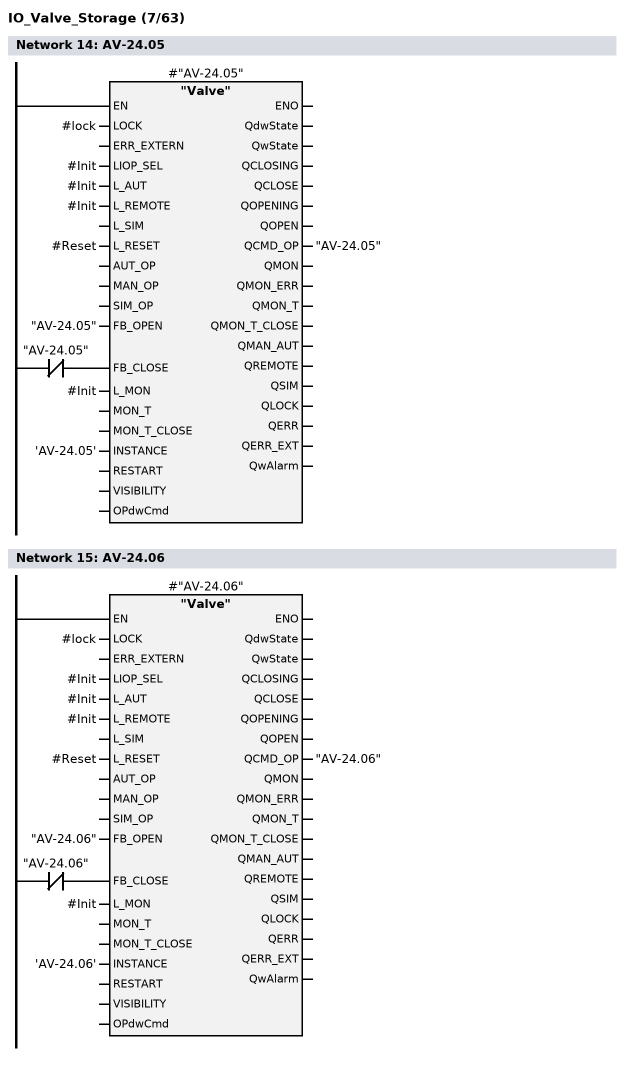
   RUNG wire#powerrail
      #"AV-24.05"(FB_CLOSE := wire#w1, LOCK := #lock, ERR_EXTERN :=, LIOP_SEL := #Init, L_AUT := #Init, L_REMOTE := #Init, L_SIM :=, L_RESET := #Reset, AUT_OP :=, MAN_OP :=, SIM_OP :=, FB_OPEN := "AV-24.05", L_MON := #Init, MON_T :=, MON_T_CLOSE :=, INSTANCE := 'AV-24.05', RESTART :=, VISIBILITY :=, OPdwCmd :=, QdwState =>, QwState =>, QCLOSING =>, QCLOSE =>, QOPENING =>, QOPEN =>, QCMD_OP => "AV-24.05", QMON =>, QMON_ERR =>, QMON_T =>, QMON_T_CLOSE =>, QMAN_AUT =>, QREMOTE =>, QSIM =>, QLOCK =>, QERR =>, QERR_EXT =>, QwAlarm =>)
   END_RUNG
   RUNG wire#powerrail
      I_Contact( "AV-24.05" )
   END_RUNG wire#w1
   // the same network as SCL:
   #"AV-24.05"(LOCK := #lock,   // "Valve"
               LIOP_SEL := #Init,
               L_AUT := #Init,
               L_REMOTE := #Init,
               L_RESET := #Reset,
               FB_OPEN := "AV-24.05",
               FB_CLOSE := NOT "AV-24.05",
               L_MON := #Init,
               INSTANCE := 'AV-24.05',
               QCMD_OP => "AV-24.05");
END_REGION

REGION Network 15: AV-24.06
   RUNG wire#powerrail
      #"AV-24.06"(FB_CLOSE := wire#w1, LOCK := #lock, ERR_EXTERN :=, LIOP_SEL := #Init, L_AUT := #Init, L_REMOTE := #Init, L_SIM :=, L_RESET := #Reset, AUT_OP :=, MAN_OP :=, SIM_OP :=, FB_OPEN := "AV-24.06", L_MON := #Init, MON_T :=, MON_T_CLOSE :=, INSTANCE := 'AV-24.06', RESTART :=, VISIBILITY :=, OPdwCmd :=, QdwState =>, QwState =>, QCLOSING =>, QCLOSE =>, QOPENING =>, QOPEN =>, QCMD_OP => "AV-24.06", QMON =>, QMON_ERR =>, QMON_T =>, QMON_T_CLOSE =>, QMAN_AUT =>, QREMOTE =>, QSIM =>, QLOCK =>, QERR =>, QERR_EXT =>, QwAlarm =>)
   END_RUNG
   RUNG wire#powerrail
      I_Contact( "AV-24.06" )
   END_RUNG wire#w1
   // the same network as SCL:
   #"AV-24.06"(LOCK := #lock,   // "Valve"
               LIOP_SEL := #Init,
               L_AUT := #Init,
               L_REMOTE := #Init,
               L_RESET := #Reset,
               FB_OPEN := "AV-24.06",
               FB_CLOSE := NOT "AV-24.06",
               L_MON := #Init,
               INSTANCE := 'AV-24.06',
               QCMD_OP => "AV-24.06");
END_REGION

REGION Network 16: AV-24.09
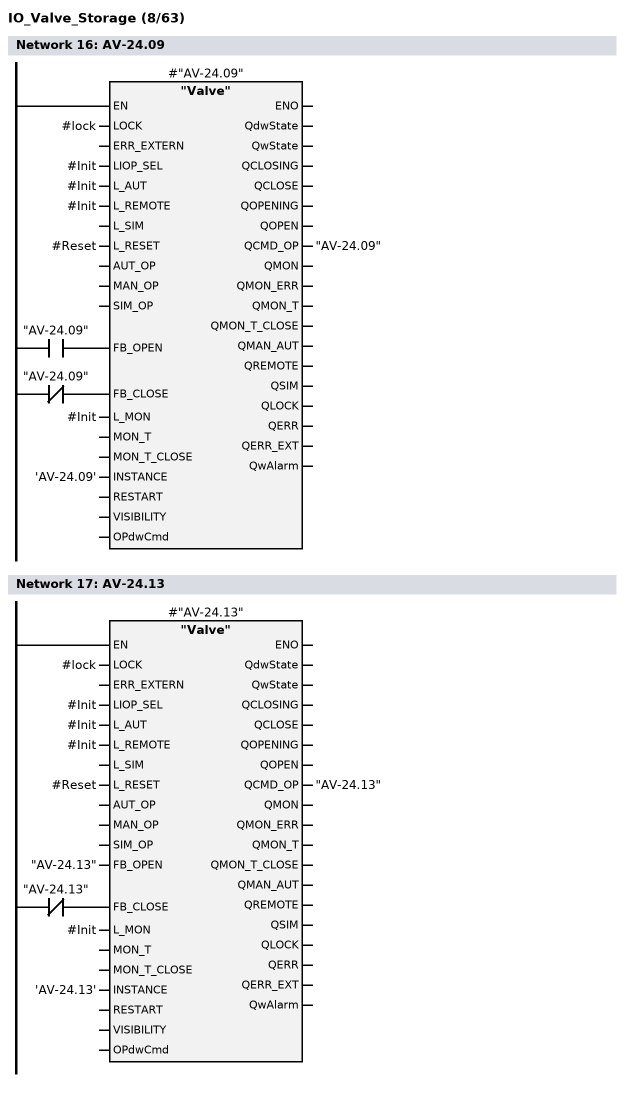
   RUNG wire#powerrail
      #"AV-24.09"(FB_OPEN := wire#w1, FB_CLOSE := wire#w2, LOCK := #lock, ERR_EXTERN :=, LIOP_SEL := #Init, L_AUT := #Init, L_REMOTE := #Init, L_SIM :=, L_RESET := #Reset, AUT_OP :=, MAN_OP :=, SIM_OP :=, L_MON := #Init, MON_T :=, MON_T_CLOSE :=, INSTANCE := 'AV-24.09', RESTART :=, VISIBILITY :=, OPdwCmd :=, QdwState =>, QwState =>, QCLOSING =>, QCLOSE =>, QOPENING =>, QOPEN =>, QCMD_OP => "AV-24.09", QMON =>, QMON_ERR =>, QMON_T =>, QMON_T_CLOSE =>, QMAN_AUT =>, QREMOTE =>, QSIM =>, QLOCK =>, QERR =>, QERR_EXT =>, QwAlarm =>)
   END_RUNG
   RUNG wire#powerrail
      Contact( "AV-24.09" )
   END_RUNG wire#w1
   RUNG wire#powerrail
      I_Contact( "AV-24.09" )
   END_RUNG wire#w2
   // the same network as SCL:
   #"AV-24.09"(LOCK := #lock,   // "Valve"
               LIOP_SEL := #Init,
               L_AUT := #Init,
               L_REMOTE := #Init,
               L_RESET := #Reset,
               FB_OPEN := "AV-24.09",
               FB_CLOSE := NOT "AV-24.09",
               L_MON := #Init,
               INSTANCE := 'AV-24.09',
               QCMD_OP => "AV-24.09");
END_REGION

REGION Network 17: AV-24.13
   RUNG wire#powerrail
      #"AV-24.13"(FB_CLOSE := wire#w1, LOCK := #lock, ERR_EXTERN :=, LIOP_SEL := #Init, L_AUT := #Init, L_REMOTE := #Init, L_SIM :=, L_RESET := #Reset, AUT_OP :=, MAN_OP :=, SIM_OP :=, FB_OPEN := "AV-24.13", L_MON := #Init, MON_T :=, MON_T_CLOSE :=, INSTANCE := 'AV-24.13', RESTART :=, VISIBILITY :=, OPdwCmd :=, QdwState =>, QwState =>, QCLOSING =>, QCLOSE =>, QOPENING =>, QOPEN =>, QCMD_OP => "AV-24.13", QMON =>, QMON_ERR =>, QMON_T =>, QMON_T_CLOSE =>, QMAN_AUT =>, QREMOTE =>, QSIM =>, QLOCK =>, QERR =>, QERR_EXT =>, QwAlarm =>)
   END_RUNG
   RUNG wire#powerrail
      I_Contact( "AV-24.13" )
   END_RUNG wire#w1
   // the same network as SCL:
   #"AV-24.13"(LOCK := #lock,   // "Valve"
               LIOP_SEL := #Init,
               L_AUT := #Init,
               L_REMOTE := #Init,
               L_RESET := #Reset,
               FB_OPEN := "AV-24.13",
               FB_CLOSE := NOT "AV-24.13",
               L_MON := #Init,
               INSTANCE := 'AV-24.13',
               QCMD_OP => "AV-24.13");
END_REGION

REGION Network 18: AV-24.14
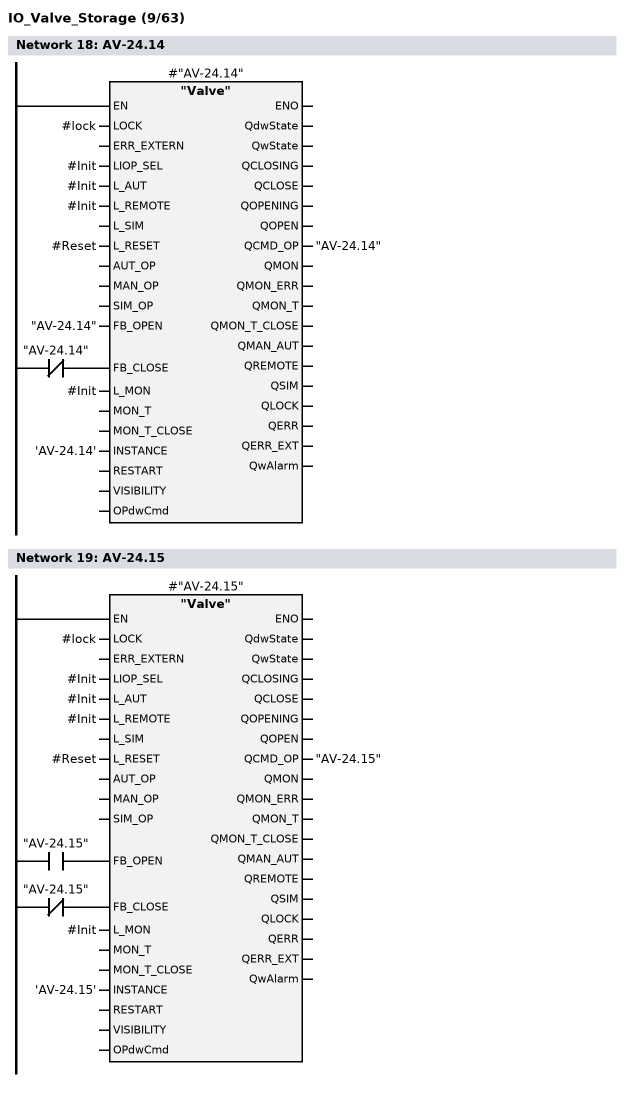
   RUNG wire#powerrail
      #"AV-24.14"(FB_CLOSE := wire#w1, LOCK := #lock, ERR_EXTERN :=, LIOP_SEL := #Init, L_AUT := #Init, L_REMOTE := #Init, L_SIM :=, L_RESET := #Reset, AUT_OP :=, MAN_OP :=, SIM_OP :=, FB_OPEN := "AV-24.14", L_MON := #Init, MON_T :=, MON_T_CLOSE :=, INSTANCE := 'AV-24.14', RESTART :=, VISIBILITY :=, OPdwCmd :=, QdwState =>, QwState =>, QCLOSING =>, QCLOSE =>, QOPENING =>, QOPEN =>, QCMD_OP => "AV-24.14", QMON =>, QMON_ERR =>, QMON_T =>, QMON_T_CLOSE =>, QMAN_AUT =>, QREMOTE =>, QSIM =>, QLOCK =>, QERR =>, QERR_EXT =>, QwAlarm =>)
   END_RUNG
   RUNG wire#powerrail
      I_Contact( "AV-24.14" )
   END_RUNG wire#w1
   // the same network as SCL:
   #"AV-24.14"(LOCK := #lock,   // "Valve"
               LIOP_SEL := #Init,
               L_AUT := #Init,
               L_REMOTE := #Init,
               L_RESET := #Reset,
               FB_OPEN := "AV-24.14",
               FB_CLOSE := NOT "AV-24.14",
               L_MON := #Init,
               INSTANCE := 'AV-24.14',
               QCMD_OP => "AV-24.14");
END_REGION

REGION Network 19: AV-24.15
   RUNG wire#powerrail
      #"AV-24.15"(FB_OPEN := wire#w1, FB_CLOSE := wire#w2, LOCK := #lock, ERR_EXTERN :=, LIOP_SEL := #Init, L_AUT := #Init, L_REMOTE := #Init, L_SIM :=, L_RESET := #Reset, AUT_OP :=, MAN_OP :=, SIM_OP :=, L_MON := #Init, MON_T :=, MON_T_CLOSE :=, INSTANCE := 'AV-24.15', RESTART :=, VISIBILITY :=, OPdwCmd :=, QdwState =>, QwState =>, QCLOSING =>, QCLOSE =>, QOPENING =>, QOPEN =>, QCMD_OP => "AV-24.15", QMON =>, QMON_ERR =>, QMON_T =>, QMON_T_CLOSE =>, QMAN_AUT =>, QREMOTE =>, QSIM =>, QLOCK =>, QERR =>, QERR_EXT =>, QwAlarm =>)
   END_RUNG
   RUNG wire#powerrail
      Contact( "AV-24.15" )
   END_RUNG wire#w1
   RUNG wire#powerrail
      I_Contact( "AV-24.15" )
   END_RUNG wire#w2
   // the same network as SCL:
   #"AV-24.15"(LOCK := #lock,   // "Valve"
               LIOP_SEL := #Init,
               L_AUT := #Init,
               L_REMOTE := #Init,
               L_RESET := #Reset,
               FB_OPEN := "AV-24.15",
               FB_CLOSE := NOT "AV-24.15",
               L_MON := #Init,
               INSTANCE := 'AV-24.15',
               QCMD_OP => "AV-24.15");
END_REGION

REGION Network 20: AV-24.16
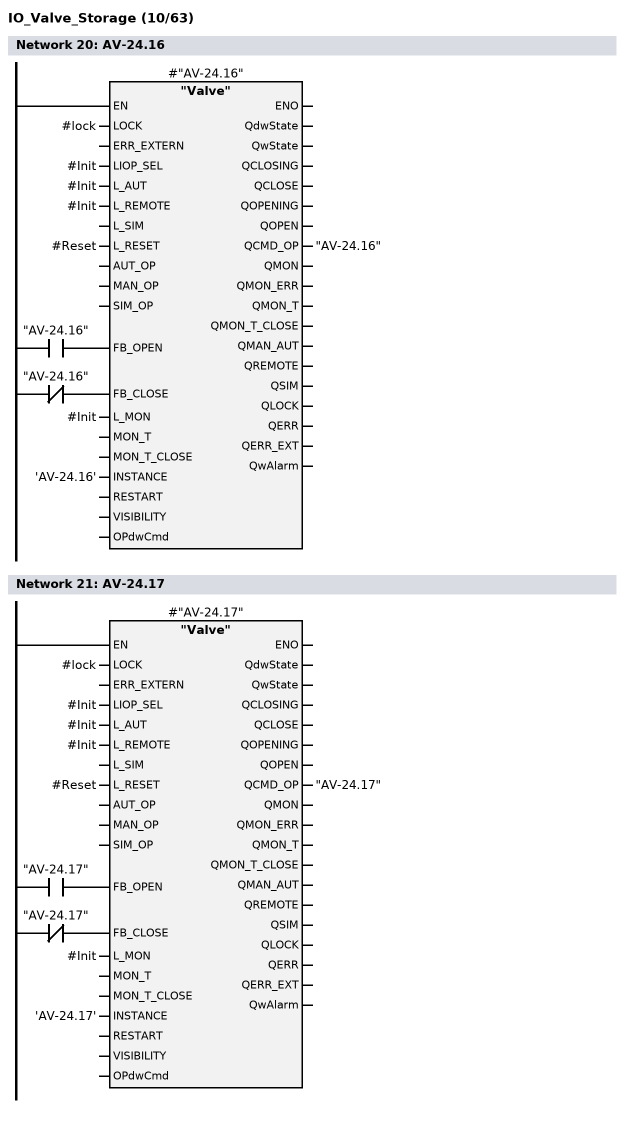
   RUNG wire#powerrail
      #"AV-24.16"(FB_OPEN := wire#w1, FB_CLOSE := wire#w2, LOCK := #lock, ERR_EXTERN :=, LIOP_SEL := #Init, L_AUT := #Init, L_REMOTE := #Init, L_SIM :=, L_RESET := #Reset, AUT_OP :=, MAN_OP :=, SIM_OP :=, L_MON := #Init, MON_T :=, MON_T_CLOSE :=, INSTANCE := 'AV-24.16', RESTART :=, VISIBILITY :=, OPdwCmd :=, QdwState =>, QwState =>, QCLOSING =>, QCLOSE =>, QOPENING =>, QOPEN =>, QCMD_OP => "AV-24.16", QMON =>, QMON_ERR =>, QMON_T =>, QMON_T_CLOSE =>, QMAN_AUT =>, QREMOTE =>, QSIM =>, QLOCK =>, QERR =>, QERR_EXT =>, QwAlarm =>)
   END_RUNG
   RUNG wire#powerrail
      Contact( "AV-24.16" )
   END_RUNG wire#w1
   RUNG wire#powerrail
      I_Contact( "AV-24.16" )
   END_RUNG wire#w2
   // the same network as SCL:
   #"AV-24.16"(LOCK := #lock,   // "Valve"
               LIOP_SEL := #Init,
               L_AUT := #Init,
               L_REMOTE := #Init,
               L_RESET := #Reset,
               FB_OPEN := "AV-24.16",
               FB_CLOSE := NOT "AV-24.16",
               L_MON := #Init,
               INSTANCE := 'AV-24.16',
               QCMD_OP => "AV-24.16");
END_REGION

REGION Network 21: AV-24.17
   RUNG wire#powerrail
      #"AV-24.17"(FB_OPEN := wire#w1, FB_CLOSE := wire#w2, LOCK := #lock, ERR_EXTERN :=, LIOP_SEL := #Init, L_AUT := #Init, L_REMOTE := #Init, L_SIM :=, L_RESET := #Reset, AUT_OP :=, MAN_OP :=, SIM_OP :=, L_MON := #Init, MON_T :=, MON_T_CLOSE :=, INSTANCE := 'AV-24.17', RESTART :=, VISIBILITY :=, OPdwCmd :=, QdwState =>, QwState =>, QCLOSING =>, QCLOSE =>, QOPENING =>, QOPEN =>, QCMD_OP => "AV-24.17", QMON =>, QMON_ERR =>, QMON_T =>, QMON_T_CLOSE =>, QMAN_AUT =>, QREMOTE =>, QSIM =>, QLOCK =>, QERR =>, QERR_EXT =>, QwAlarm =>)
   END_RUNG
   RUNG wire#powerrail
      Contact( "AV-24.17" )
   END_RUNG wire#w1
   RUNG wire#powerrail
      I_Contact( "AV-24.17" )
   END_RUNG wire#w2
   // the same network as SCL:
   #"AV-24.17"(LOCK := #lock,   // "Valve"
               LIOP_SEL := #Init,
               L_AUT := #Init,
               L_REMOTE := #Init,
               L_RESET := #Reset,
               FB_OPEN := "AV-24.17",
               FB_CLOSE := NOT "AV-24.17",
               L_MON := #Init,
               INSTANCE := 'AV-24.17',
               QCMD_OP => "AV-24.17");
END_REGION

REGION Network 22: AV-24.18
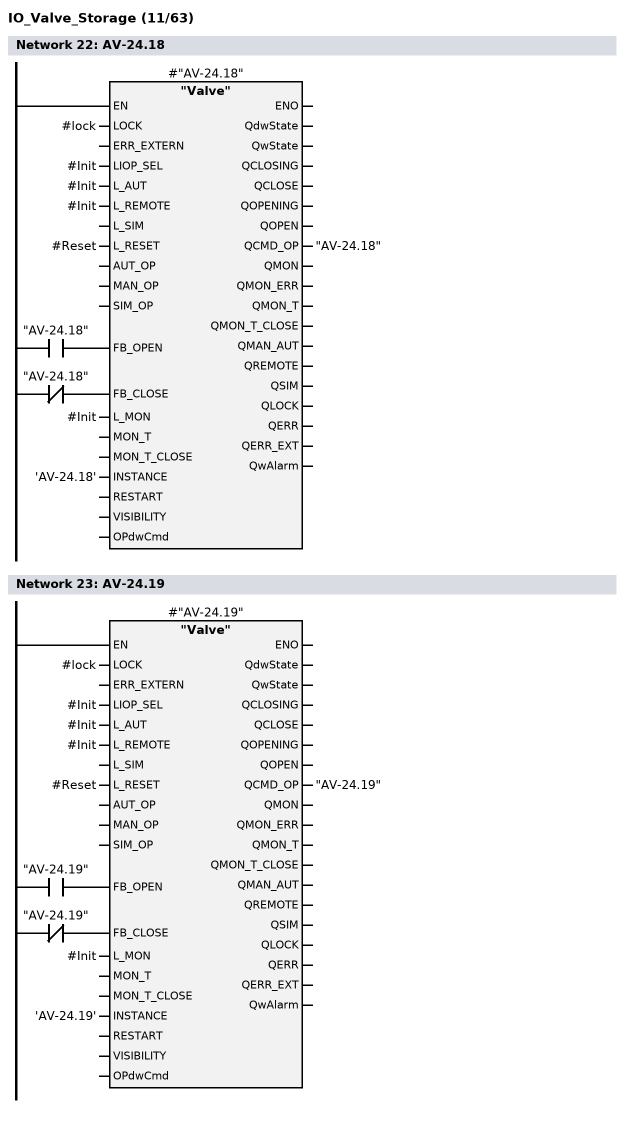
   RUNG wire#powerrail
      #"AV-24.18"(FB_OPEN := wire#w1, FB_CLOSE := wire#w2, LOCK := #lock, ERR_EXTERN :=, LIOP_SEL := #Init, L_AUT := #Init, L_REMOTE := #Init, L_SIM :=, L_RESET := #Reset, AUT_OP :=, MAN_OP :=, SIM_OP :=, L_MON := #Init, MON_T :=, MON_T_CLOSE :=, INSTANCE := 'AV-24.18', RESTART :=, VISIBILITY :=, OPdwCmd :=, QdwState =>, QwState =>, QCLOSING =>, QCLOSE =>, QOPENING =>, QOPEN =>, QCMD_OP => "AV-24.18", QMON =>, QMON_ERR =>, QMON_T =>, QMON_T_CLOSE =>, QMAN_AUT =>, QREMOTE =>, QSIM =>, QLOCK =>, QERR =>, QERR_EXT =>, QwAlarm =>)
   END_RUNG
   RUNG wire#powerrail
      Contact( "AV-24.18" )
   END_RUNG wire#w1
   RUNG wire#powerrail
      I_Contact( "AV-24.18" )
   END_RUNG wire#w2
   // the same network as SCL:
   #"AV-24.18"(LOCK := #lock,   // "Valve"
               LIOP_SEL := #Init,
               L_AUT := #Init,
               L_REMOTE := #Init,
               L_RESET := #Reset,
               FB_OPEN := "AV-24.18",
               FB_CLOSE := NOT "AV-24.18",
               L_MON := #Init,
               INSTANCE := 'AV-24.18',
               QCMD_OP => "AV-24.18");
END_REGION

REGION Network 23: AV-24.19
   RUNG wire#powerrail
      #"AV-24.19"(FB_OPEN := wire#w1, FB_CLOSE := wire#w2, LOCK := #lock, ERR_EXTERN :=, LIOP_SEL := #Init, L_AUT := #Init, L_REMOTE := #Init, L_SIM :=, L_RESET := #Reset, AUT_OP :=, MAN_OP :=, SIM_OP :=, L_MON := #Init, MON_T :=, MON_T_CLOSE :=, INSTANCE := 'AV-24.19', RESTART :=, VISIBILITY :=, OPdwCmd :=, QdwState =>, QwState =>, QCLOSING =>, QCLOSE =>, QOPENING =>, QOPEN =>, QCMD_OP => "AV-24.19", QMON =>, QMON_ERR =>, QMON_T =>, QMON_T_CLOSE =>, QMAN_AUT =>, QREMOTE =>, QSIM =>, QLOCK =>, QERR =>, QERR_EXT =>, QwAlarm =>)
   END_RUNG
   RUNG wire#powerrail
      Contact( "AV-24.19" )
   END_RUNG wire#w1
   RUNG wire#powerrail
      I_Contact( "AV-24.19" )
   END_RUNG wire#w2
   // the same network as SCL:
   #"AV-24.19"(LOCK := #lock,   // "Valve"
               LIOP_SEL := #Init,
               L_AUT := #Init,
               L_REMOTE := #Init,
               L_RESET := #Reset,
               FB_OPEN := "AV-24.19",
               FB_CLOSE := NOT "AV-24.19",
               L_MON := #Init,
               INSTANCE := 'AV-24.19',
               QCMD_OP => "AV-24.19");
END_REGION

REGION Network 24: AV-24.20
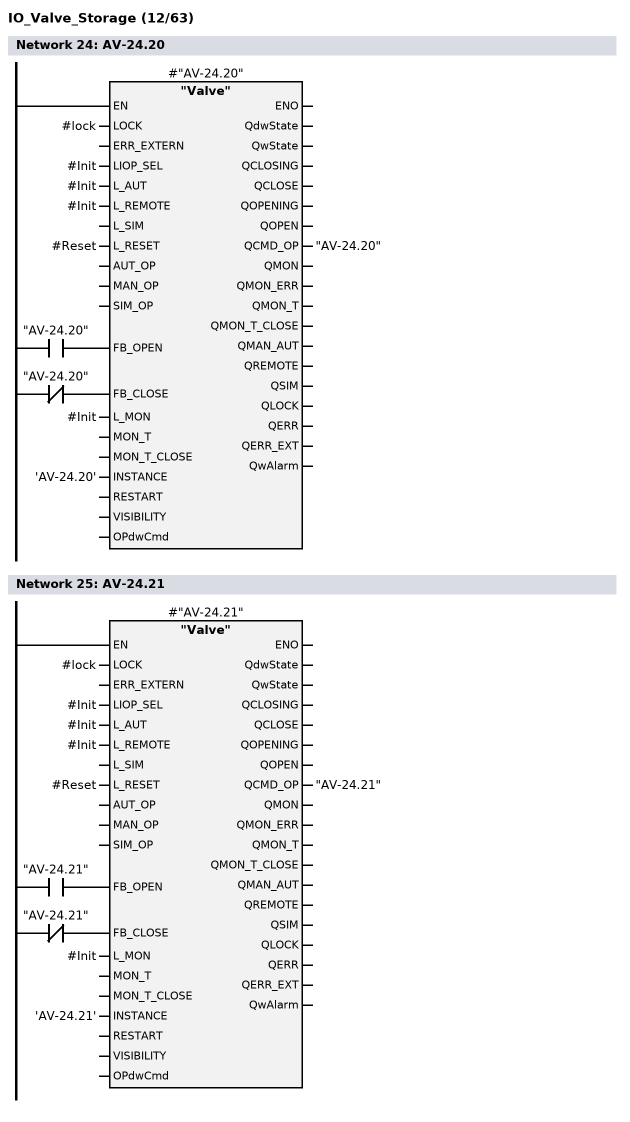
   RUNG wire#powerrail
      #"AV-24.20"(FB_OPEN := wire#w1, FB_CLOSE := wire#w2, LOCK := #lock, ERR_EXTERN :=, LIOP_SEL := #Init, L_AUT := #Init, L_REMOTE := #Init, L_SIM :=, L_RESET := #Reset, AUT_OP :=, MAN_OP :=, SIM_OP :=, L_MON := #Init, MON_T :=, MON_T_CLOSE :=, INSTANCE := 'AV-24.20', RESTART :=, VISIBILITY :=, OPdwCmd :=, QdwState =>, QwState =>, QCLOSING =>, QCLOSE =>, QOPENING =>, QOPEN =>, QCMD_OP => "AV-24.20", QMON =>, QMON_ERR =>, QMON_T =>, QMON_T_CLOSE =>, QMAN_AUT =>, QREMOTE =>, QSIM =>, QLOCK =>, QERR =>, QERR_EXT =>, QwAlarm =>)
   END_RUNG
   RUNG wire#powerrail
      Contact( "AV-24.20" )
   END_RUNG wire#w1
   RUNG wire#powerrail
      I_Contact( "AV-24.20" )
   END_RUNG wire#w2
   // the same network as SCL:
   #"AV-24.20"(LOCK := #lock,   // "Valve"
               LIOP_SEL := #Init,
               L_AUT := #Init,
               L_REMOTE := #Init,
               L_RESET := #Reset,
               FB_OPEN := "AV-24.20",
               FB_CLOSE := NOT "AV-24.20",
               L_MON := #Init,
               INSTANCE := 'AV-24.20',
               QCMD_OP => "AV-24.20");
END_REGION

REGION Network 25: AV-24.21
   RUNG wire#powerrail
      #"AV-24.21"(FB_OPEN := wire#w1, FB_CLOSE := wire#w2, LOCK := #lock, ERR_EXTERN :=, LIOP_SEL := #Init, L_AUT := #Init, L_REMOTE := #Init, L_SIM :=, L_RESET := #Reset, AUT_OP :=, MAN_OP :=, SIM_OP :=, L_MON := #Init, MON_T :=, MON_T_CLOSE :=, INSTANCE := 'AV-24.21', RESTART :=, VISIBILITY :=, OPdwCmd :=, QdwState =>, QwState =>, QCLOSING =>, QCLOSE =>, QOPENING =>, QOPEN =>, QCMD_OP => "AV-24.21", QMON =>, QMON_ERR =>, QMON_T =>, QMON_T_CLOSE =>, QMAN_AUT =>, QREMOTE =>, QSIM =>, QLOCK =>, QERR =>, QERR_EXT =>, QwAlarm =>)
   END_RUNG
   RUNG wire#powerrail
      Contact( "AV-24.21" )
   END_RUNG wire#w1
   RUNG wire#powerrail
      I_Contact( "AV-24.21" )
   END_RUNG wire#w2
   // the same network as SCL:
   #"AV-24.21"(LOCK := #lock,   // "Valve"
               LIOP_SEL := #Init,
               L_AUT := #Init,
               L_REMOTE := #Init,
               L_RESET := #Reset,
               FB_OPEN := "AV-24.21",
               FB_CLOSE := NOT "AV-24.21",
               L_MON := #Init,
               INSTANCE := 'AV-24.21',
               QCMD_OP => "AV-24.21");
END_REGION

REGION Network 26: AV-24.22
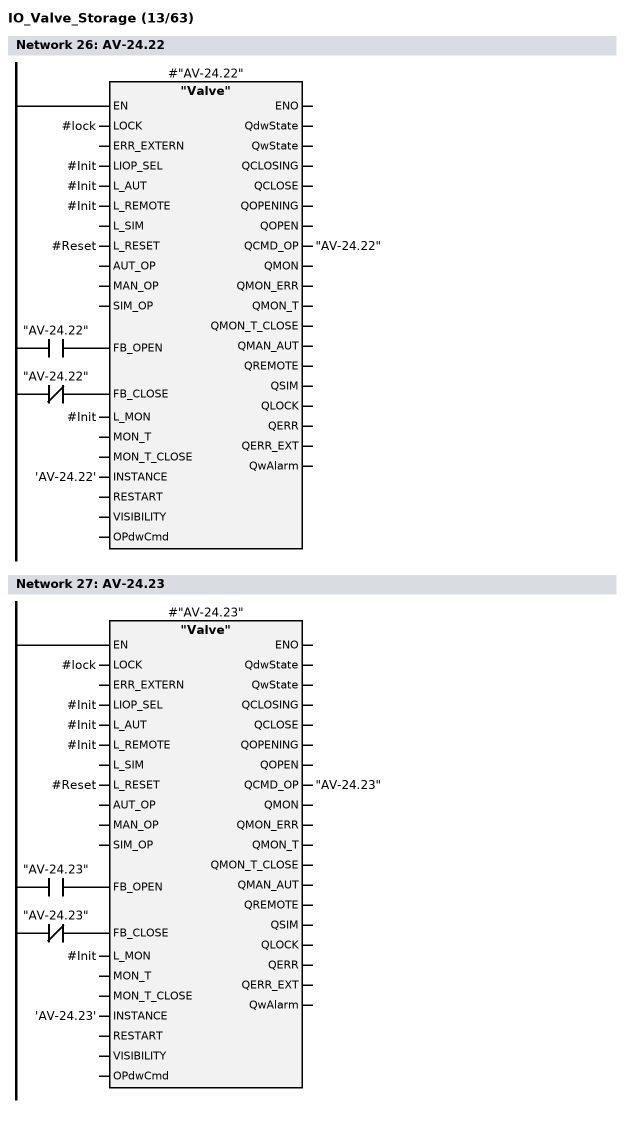
   RUNG wire#powerrail
      #"AV-24.22"(FB_OPEN := wire#w1, FB_CLOSE := wire#w2, LOCK := #lock, ERR_EXTERN :=, LIOP_SEL := #Init, L_AUT := #Init, L_REMOTE := #Init, L_SIM :=, L_RESET := #Reset, AUT_OP :=, MAN_OP :=, SIM_OP :=, L_MON := #Init, MON_T :=, MON_T_CLOSE :=, INSTANCE := 'AV-24.22', RESTART :=, VISIBILITY :=, OPdwCmd :=, QdwState =>, QwState =>, QCLOSING =>, QCLOSE =>, QOPENING =>, QOPEN =>, QCMD_OP => "AV-24.22", QMON =>, QMON_ERR =>, QMON_T =>, QMON_T_CLOSE =>, QMAN_AUT =>, QREMOTE =>, QSIM =>, QLOCK =>, QERR =>, QERR_EXT =>, QwAlarm =>)
   END_RUNG
   RUNG wire#powerrail
      Contact( "AV-24.22" )
   END_RUNG wire#w1
   RUNG wire#powerrail
      I_Contact( "AV-24.22" )
   END_RUNG wire#w2
   // the same network as SCL:
   #"AV-24.22"(LOCK := #lock,   // "Valve"
               LIOP_SEL := #Init,
               L_AUT := #Init,
               L_REMOTE := #Init,
               L_RESET := #Reset,
               FB_OPEN := "AV-24.22",
               FB_CLOSE := NOT "AV-24.22",
               L_MON := #Init,
               INSTANCE := 'AV-24.22',
               QCMD_OP => "AV-24.22");
END_REGION

REGION Network 27: AV-24.23
   RUNG wire#powerrail
      #"AV-24.23"(FB_OPEN := wire#w1, FB_CLOSE := wire#w2, LOCK := #lock, ERR_EXTERN :=, LIOP_SEL := #Init, L_AUT := #Init, L_REMOTE := #Init, L_SIM :=, L_RESET := #Reset, AUT_OP :=, MAN_OP :=, SIM_OP :=, L_MON := #Init, MON_T :=, MON_T_CLOSE :=, INSTANCE := 'AV-24.23', RESTART :=, VISIBILITY :=, OPdwCmd :=, QdwState =>, QwState =>, QCLOSING =>, QCLOSE =>, QOPENING =>, QOPEN =>, QCMD_OP => "AV-24.23", QMON =>, QMON_ERR =>, QMON_T =>, QMON_T_CLOSE =>, QMAN_AUT =>, QREMOTE =>, QSIM =>, QLOCK =>, QERR =>, QERR_EXT =>, QwAlarm =>)
   END_RUNG
   RUNG wire#powerrail
      Contact( "AV-24.23" )
   END_RUNG wire#w1
   RUNG wire#powerrail
      I_Contact( "AV-24.23" )
   END_RUNG wire#w2
   // the same network as SCL:
   #"AV-24.23"(LOCK := #lock,   // "Valve"
               LIOP_SEL := #Init,
               L_AUT := #Init,
               L_REMOTE := #Init,
               L_RESET := #Reset,
               FB_OPEN := "AV-24.23",
               FB_CLOSE := NOT "AV-24.23",
               L_MON := #Init,
               INSTANCE := 'AV-24.23',
               QCMD_OP => "AV-24.23");
END_REGION

REGION Network 28: AV-24.24
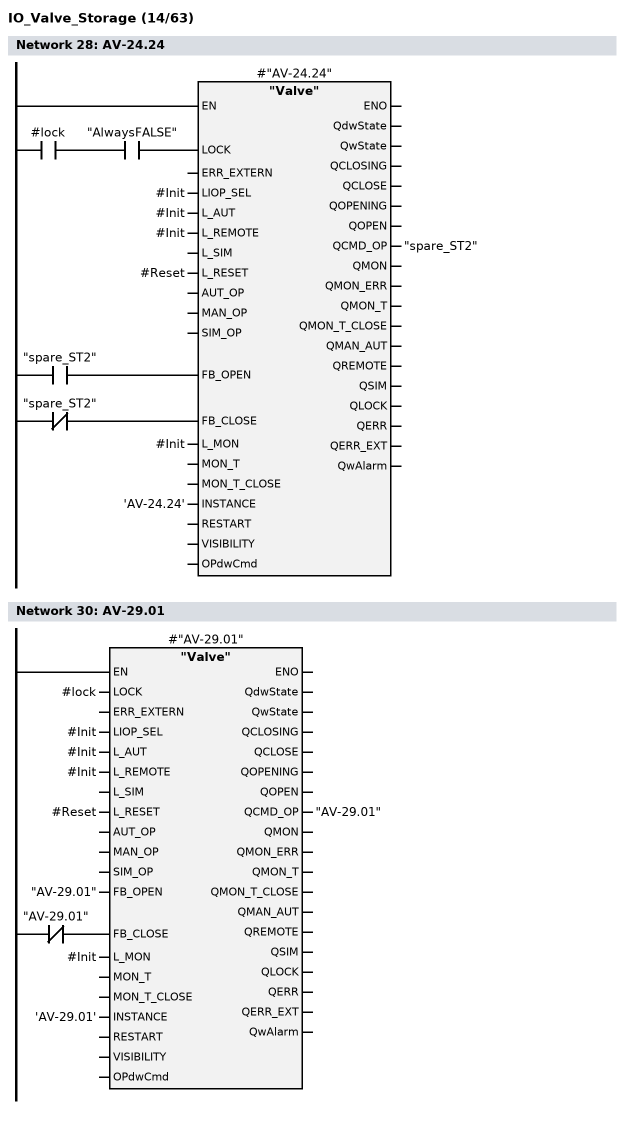
   RUNG wire#powerrail
      #"AV-24.24"(LOCK := wire#w1, FB_OPEN := wire#w2, FB_CLOSE := wire#w3, ERR_EXTERN :=, LIOP_SEL := #Init, L_AUT := #Init, L_REMOTE := #Init, L_SIM :=, L_RESET := #Reset, AUT_OP :=, MAN_OP :=, SIM_OP :=, L_MON := #Init, MON_T :=, MON_T_CLOSE :=, INSTANCE := 'AV-24.24', RESTART :=, VISIBILITY :=, OPdwCmd :=, QdwState =>, QwState =>, QCLOSING =>, QCLOSE =>, QOPENING =>, QOPEN =>, QCMD_OP => "spare_ST2", QMON =>, QMON_ERR =>, QMON_T =>, QMON_T_CLOSE =>, QMAN_AUT =>, QREMOTE =>, QSIM =>, QLOCK =>, QERR =>, QERR_EXT =>, QwAlarm =>)
   END_RUNG
   RUNG wire#powerrail
      Contact( #lock )
      Contact( "AlwaysFALSE" )
   END_RUNG wire#w1
   RUNG wire#powerrail
      Contact( "spare_ST2" )
   END_RUNG wire#w2
   RUNG wire#powerrail
      I_Contact( "spare_ST2" )
   END_RUNG wire#w3
   // the same network as SCL:
   #"AV-24.24"(LOCK := #lock AND "AlwaysFALSE",   // "Valve"
               LIOP_SEL := #Init,
               L_AUT := #Init,
               L_REMOTE := #Init,
               L_RESET := #Reset,
               FB_OPEN := "spare_ST2",
               FB_CLOSE := NOT "spare_ST2",
               L_MON := #Init,
               INSTANCE := 'AV-24.24',
               QCMD_OP => "spare_ST2");
END_REGION

REGION Network 30: AV-29.01
   RUNG wire#powerrail
      #"AV-29.01"(FB_CLOSE := wire#w1, LOCK := #lock, ERR_EXTERN :=, LIOP_SEL := #Init, L_AUT := #Init, L_REMOTE := #Init, L_SIM :=, L_RESET := #Reset, AUT_OP :=, MAN_OP :=, SIM_OP :=, FB_OPEN := "AV-29.01", L_MON := #Init, MON_T :=, MON_T_CLOSE :=, INSTANCE := 'AV-29.01', RESTART :=, VISIBILITY :=, OPdwCmd :=, QdwState =>, QwState =>, QCLOSING =>, QCLOSE =>, QOPENING =>, QOPEN =>, QCMD_OP => "AV-29.01", QMON =>, QMON_ERR =>, QMON_T =>, QMON_T_CLOSE =>, QMAN_AUT =>, QREMOTE =>, QSIM =>, QLOCK =>, QERR =>, QERR_EXT =>, QwAlarm =>)
   END_RUNG
   RUNG wire#powerrail
      I_Contact( "AV-29.01" )
   END_RUNG wire#w1
   // the same network as SCL:
   #"AV-29.01"(LOCK := #lock,   // "Valve"
               LIOP_SEL := #Init,
               L_AUT := #Init,
               L_REMOTE := #Init,
               L_RESET := #Reset,
               FB_OPEN := "AV-29.01",
               FB_CLOSE := NOT "AV-29.01",
               L_MON := #Init,
               INSTANCE := 'AV-29.01',
               QCMD_OP => "AV-29.01");
END_REGION

REGION Network 31: AV-29.02
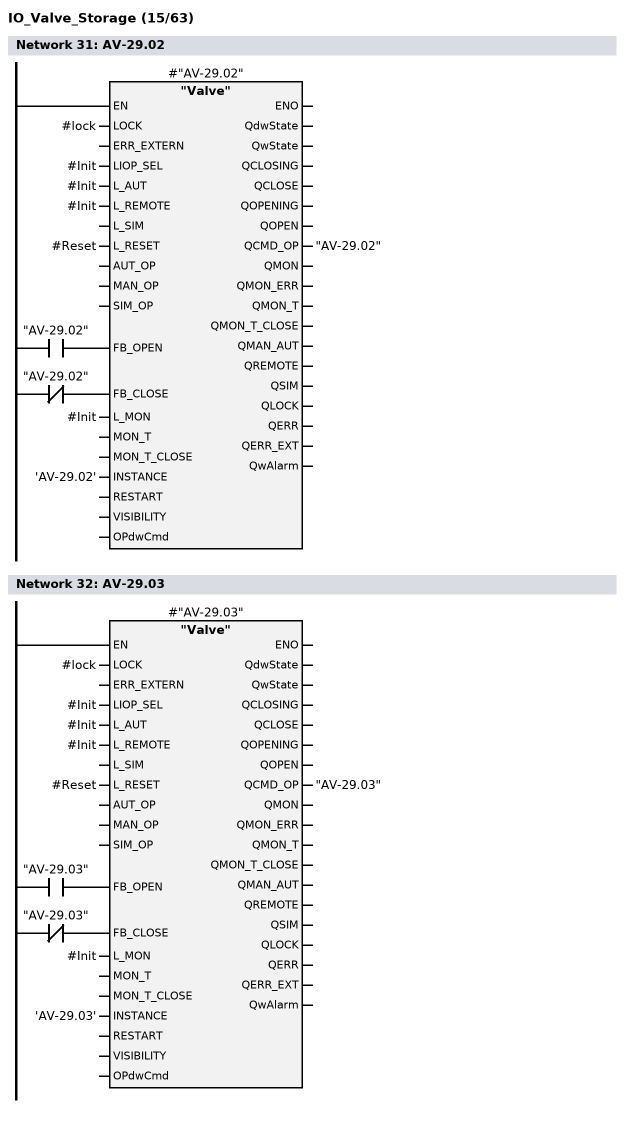
   RUNG wire#powerrail
      #"AV-29.02"(FB_OPEN := wire#w1, FB_CLOSE := wire#w2, LOCK := #lock, ERR_EXTERN :=, LIOP_SEL := #Init, L_AUT := #Init, L_REMOTE := #Init, L_SIM :=, L_RESET := #Reset, AUT_OP :=, MAN_OP :=, SIM_OP :=, L_MON := #Init, MON_T :=, MON_T_CLOSE :=, INSTANCE := 'AV-29.02', RESTART :=, VISIBILITY :=, OPdwCmd :=, QdwState =>, QwState =>, QCLOSING =>, QCLOSE =>, QOPENING =>, QOPEN =>, QCMD_OP => "AV-29.02", QMON =>, QMON_ERR =>, QMON_T =>, QMON_T_CLOSE =>, QMAN_AUT =>, QREMOTE =>, QSIM =>, QLOCK =>, QERR =>, QERR_EXT =>, QwAlarm =>)
   END_RUNG
   RUNG wire#powerrail
      Contact( "AV-29.02" )
   END_RUNG wire#w1
   RUNG wire#powerrail
      I_Contact( "AV-29.02" )
   END_RUNG wire#w2
   // the same network as SCL:
   #"AV-29.02"(LOCK := #lock,   // "Valve"
               LIOP_SEL := #Init,
               L_AUT := #Init,
               L_REMOTE := #Init,
               L_RESET := #Reset,
               FB_OPEN := "AV-29.02",
               FB_CLOSE := NOT "AV-29.02",
               L_MON := #Init,
               INSTANCE := 'AV-29.02',
               QCMD_OP => "AV-29.02");
END_REGION

REGION Network 32: AV-29.03
   RUNG wire#powerrail
      #"AV-29.03"(FB_OPEN := wire#w1, FB_CLOSE := wire#w2, LOCK := #lock, ERR_EXTERN :=, LIOP_SEL := #Init, L_AUT := #Init, L_REMOTE := #Init, L_SIM :=, L_RESET := #Reset, AUT_OP :=, MAN_OP :=, SIM_OP :=, L_MON := #Init, MON_T :=, MON_T_CLOSE :=, INSTANCE := 'AV-29.03', RESTART :=, VISIBILITY :=, OPdwCmd :=, QdwState =>, QwState =>, QCLOSING =>, QCLOSE =>, QOPENING =>, QOPEN =>, QCMD_OP => "AV-29.03", QMON =>, QMON_ERR =>, QMON_T =>, QMON_T_CLOSE =>, QMAN_AUT =>, QREMOTE =>, QSIM =>, QLOCK =>, QERR =>, QERR_EXT =>, QwAlarm =>)
   END_RUNG
   RUNG wire#powerrail
      Contact( "AV-29.03" )
   END_RUNG wire#w1
   RUNG wire#powerrail
      I_Contact( "AV-29.03" )
   END_RUNG wire#w2
   // the same network as SCL:
   #"AV-29.03"(LOCK := #lock,   // "Valve"
               LIOP_SEL := #Init,
               L_AUT := #Init,
               L_REMOTE := #Init,
               L_RESET := #Reset,
               FB_OPEN := "AV-29.03",
               FB_CLOSE := NOT "AV-29.03",
               L_MON := #Init,
               INSTANCE := 'AV-29.03',
               QCMD_OP => "AV-29.03");
END_REGION

REGION Network 33: AV-29.04
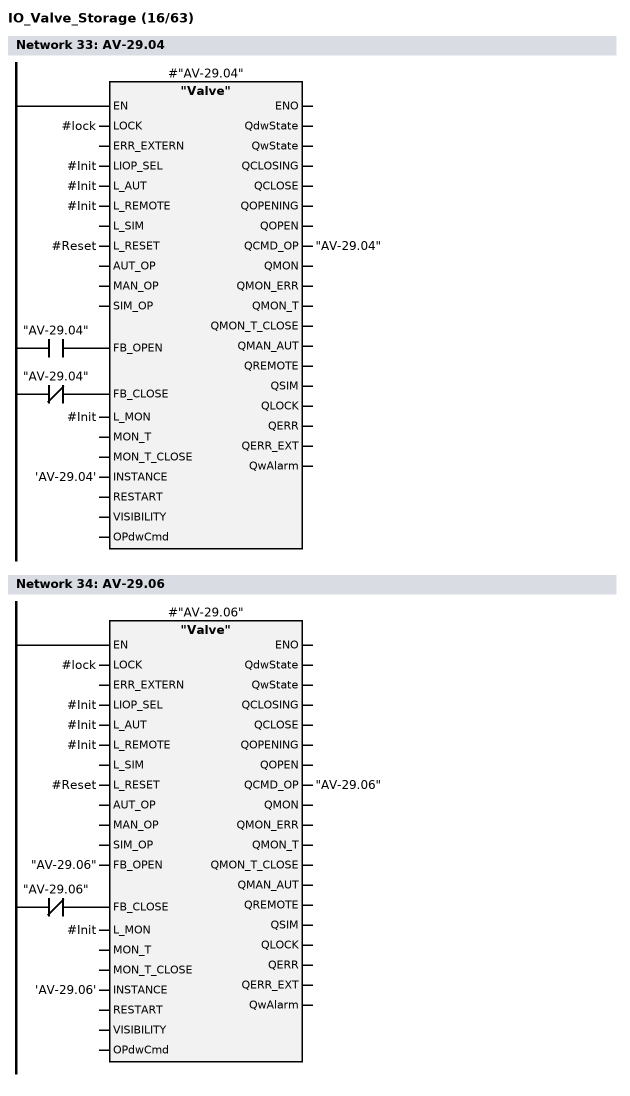
   RUNG wire#powerrail
      #"AV-29.04"(FB_OPEN := wire#w1, FB_CLOSE := wire#w2, LOCK := #lock, ERR_EXTERN :=, LIOP_SEL := #Init, L_AUT := #Init, L_REMOTE := #Init, L_SIM :=, L_RESET := #Reset, AUT_OP :=, MAN_OP :=, SIM_OP :=, L_MON := #Init, MON_T :=, MON_T_CLOSE :=, INSTANCE := 'AV-29.04', RESTART :=, VISIBILITY :=, OPdwCmd :=, QdwState =>, QwState =>, QCLOSING =>, QCLOSE =>, QOPENING =>, QOPEN =>, QCMD_OP => "AV-29.04", QMON =>, QMON_ERR =>, QMON_T =>, QMON_T_CLOSE =>, QMAN_AUT =>, QREMOTE =>, QSIM =>, QLOCK =>, QERR =>, QERR_EXT =>, QwAlarm =>)
   END_RUNG
   RUNG wire#powerrail
      Contact( "AV-29.04" )
   END_RUNG wire#w1
   RUNG wire#powerrail
      I_Contact( "AV-29.04" )
   END_RUNG wire#w2
   // the same network as SCL:
   #"AV-29.04"(LOCK := #lock,   // "Valve"
               LIOP_SEL := #Init,
               L_AUT := #Init,
               L_REMOTE := #Init,
               L_RESET := #Reset,
               FB_OPEN := "AV-29.04",
               FB_CLOSE := NOT "AV-29.04",
               L_MON := #Init,
               INSTANCE := 'AV-29.04',
               QCMD_OP => "AV-29.04");
END_REGION

REGION Network 34: AV-29.06
   RUNG wire#powerrail
      #"AV-29.06"(FB_CLOSE := wire#w1, LOCK := #lock, ERR_EXTERN :=, LIOP_SEL := #Init, L_AUT := #Init, L_REMOTE := #Init, L_SIM :=, L_RESET := #Reset, AUT_OP :=, MAN_OP :=, SIM_OP :=, FB_OPEN := "AV-29.06", L_MON := #Init, MON_T :=, MON_T_CLOSE :=, INSTANCE := 'AV-29.06', RESTART :=, VISIBILITY :=, OPdwCmd :=, QdwState =>, QwState =>, QCLOSING =>, QCLOSE =>, QOPENING =>, QOPEN =>, QCMD_OP => "AV-29.06", QMON =>, QMON_ERR =>, QMON_T =>, QMON_T_CLOSE =>, QMAN_AUT =>, QREMOTE =>, QSIM =>, QLOCK =>, QERR =>, QERR_EXT =>, QwAlarm =>)
   END_RUNG
   RUNG wire#powerrail
      I_Contact( "AV-29.06" )
   END_RUNG wire#w1
   // the same network as SCL:
   #"AV-29.06"(LOCK := #lock,   // "Valve"
               LIOP_SEL := #Init,
               L_AUT := #Init,
               L_REMOTE := #Init,
               L_RESET := #Reset,
               FB_OPEN := "AV-29.06",
               FB_CLOSE := NOT "AV-29.06",
               L_MON := #Init,
               INSTANCE := 'AV-29.06',
               QCMD_OP => "AV-29.06");
END_REGION

REGION Network 36: AV-33.01
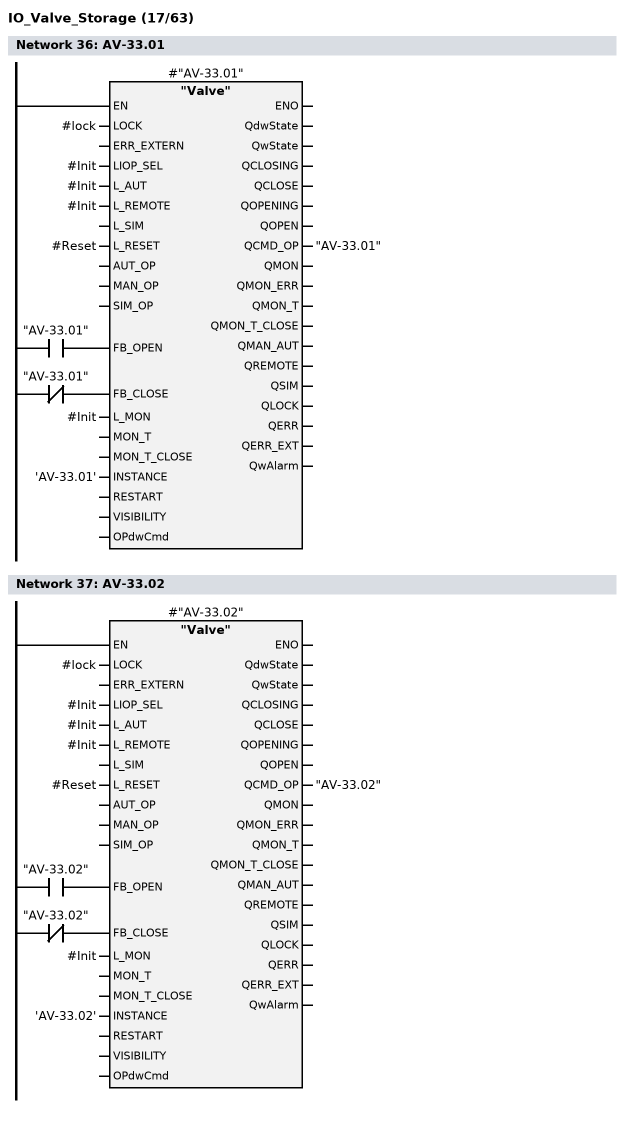
   RUNG wire#powerrail
      #"AV-33.01"(FB_OPEN := wire#w1, FB_CLOSE := wire#w2, LOCK := #lock, ERR_EXTERN :=, LIOP_SEL := #Init, L_AUT := #Init, L_REMOTE := #Init, L_SIM :=, L_RESET := #Reset, AUT_OP :=, MAN_OP :=, SIM_OP :=, L_MON := #Init, MON_T :=, MON_T_CLOSE :=, INSTANCE := 'AV-33.01', RESTART :=, VISIBILITY :=, OPdwCmd :=, QdwState =>, QwState =>, QCLOSING =>, QCLOSE =>, QOPENING =>, QOPEN =>, QCMD_OP => "AV-33.01", QMON =>, QMON_ERR =>, QMON_T =>, QMON_T_CLOSE =>, QMAN_AUT =>, QREMOTE =>, QSIM =>, QLOCK =>, QERR =>, QERR_EXT =>, QwAlarm =>)
   END_RUNG
   RUNG wire#powerrail
      Contact( "AV-33.01" )
   END_RUNG wire#w1
   RUNG wire#powerrail
      I_Contact( "AV-33.01" )
   END_RUNG wire#w2
   // the same network as SCL:
   #"AV-33.01"(LOCK := #lock,   // "Valve"
               LIOP_SEL := #Init,
               L_AUT := #Init,
               L_REMOTE := #Init,
               L_RESET := #Reset,
               FB_OPEN := "AV-33.01",
               FB_CLOSE := NOT "AV-33.01",
               L_MON := #Init,
               INSTANCE := 'AV-33.01',
               QCMD_OP => "AV-33.01");
END_REGION

REGION Network 37: AV-33.02
   RUNG wire#powerrail
      #"AV-33.02"(FB_OPEN := wire#w1, FB_CLOSE := wire#w2, LOCK := #lock, ERR_EXTERN :=, LIOP_SEL := #Init, L_AUT := #Init, L_REMOTE := #Init, L_SIM :=, L_RESET := #Reset, AUT_OP :=, MAN_OP :=, SIM_OP :=, L_MON := #Init, MON_T :=, MON_T_CLOSE :=, INSTANCE := 'AV-33.02', RESTART :=, VISIBILITY :=, OPdwCmd :=, QdwState =>, QwState =>, QCLOSING =>, QCLOSE =>, QOPENING =>, QOPEN =>, QCMD_OP => "AV-33.02", QMON =>, QMON_ERR =>, QMON_T =>, QMON_T_CLOSE =>, QMAN_AUT =>, QREMOTE =>, QSIM =>, QLOCK =>, QERR =>, QERR_EXT =>, QwAlarm =>)
   END_RUNG
   RUNG wire#powerrail
      Contact( "AV-33.02" )
   END_RUNG wire#w1
   RUNG wire#powerrail
      I_Contact( "AV-33.02" )
   END_RUNG wire#w2
   // the same network as SCL:
   #"AV-33.02"(LOCK := #lock,   // "Valve"
               LIOP_SEL := #Init,
               L_AUT := #Init,
               L_REMOTE := #Init,
               L_RESET := #Reset,
               FB_OPEN := "AV-33.02",
               FB_CLOSE := NOT "AV-33.02",
               L_MON := #Init,
               INSTANCE := 'AV-33.02',
               QCMD_OP => "AV-33.02");
END_REGION

REGION Network 38: AV-33.03
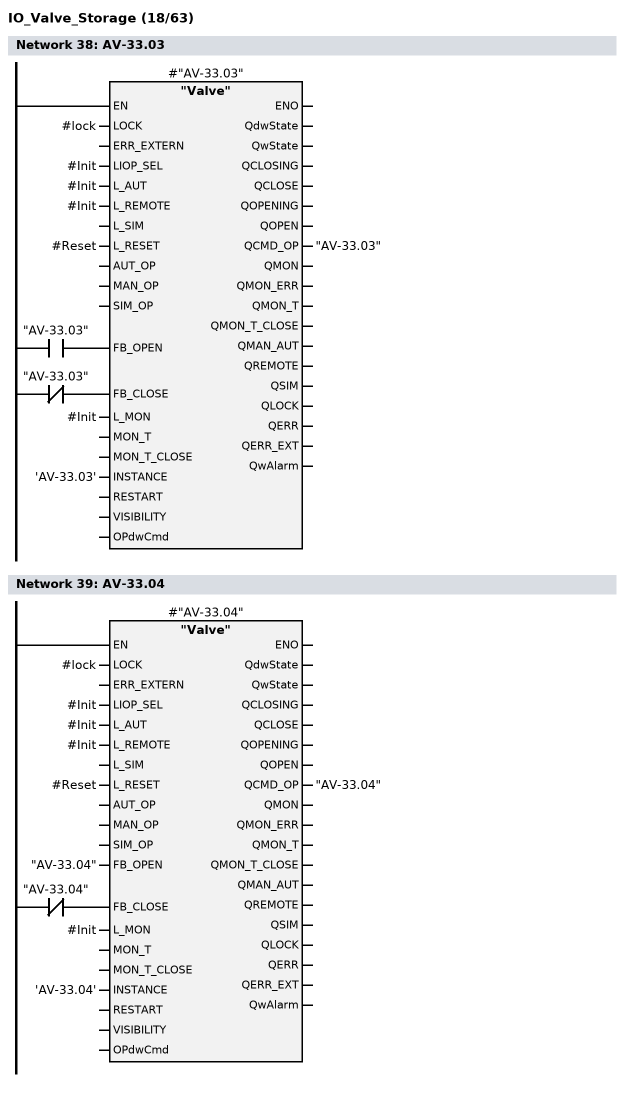
   RUNG wire#powerrail
      #"AV-33.03"(FB_OPEN := wire#w1, FB_CLOSE := wire#w2, LOCK := #lock, ERR_EXTERN :=, LIOP_SEL := #Init, L_AUT := #Init, L_REMOTE := #Init, L_SIM :=, L_RESET := #Reset, AUT_OP :=, MAN_OP :=, SIM_OP :=, L_MON := #Init, MON_T :=, MON_T_CLOSE :=, INSTANCE := 'AV-33.03', RESTART :=, VISIBILITY :=, OPdwCmd :=, QdwState =>, QwState =>, QCLOSING =>, QCLOSE =>, QOPENING =>, QOPEN =>, QCMD_OP => "AV-33.03", QMON =>, QMON_ERR =>, QMON_T =>, QMON_T_CLOSE =>, QMAN_AUT =>, QREMOTE =>, QSIM =>, QLOCK =>, QERR =>, QERR_EXT =>, QwAlarm =>)
   END_RUNG
   RUNG wire#powerrail
      Contact( "AV-33.03" )
   END_RUNG wire#w1
   RUNG wire#powerrail
      I_Contact( "AV-33.03" )
   END_RUNG wire#w2
   // the same network as SCL:
   #"AV-33.03"(LOCK := #lock,   // "Valve"
               LIOP_SEL := #Init,
               L_AUT := #Init,
               L_REMOTE := #Init,
               L_RESET := #Reset,
               FB_OPEN := "AV-33.03",
               FB_CLOSE := NOT "AV-33.03",
               L_MON := #Init,
               INSTANCE := 'AV-33.03',
               QCMD_OP => "AV-33.03");
END_REGION

REGION Network 39: AV-33.04
   RUNG wire#powerrail
      #"AV-33.04"(FB_CLOSE := wire#w1, LOCK := #lock, ERR_EXTERN :=, LIOP_SEL := #Init, L_AUT := #Init, L_REMOTE := #Init, L_SIM :=, L_RESET := #Reset, AUT_OP :=, MAN_OP :=, SIM_OP :=, FB_OPEN := "AV-33.04", L_MON := #Init, MON_T :=, MON_T_CLOSE :=, INSTANCE := 'AV-33.04', RESTART :=, VISIBILITY :=, OPdwCmd :=, QdwState =>, QwState =>, QCLOSING =>, QCLOSE =>, QOPENING =>, QOPEN =>, QCMD_OP => "AV-33.04", QMON =>, QMON_ERR =>, QMON_T =>, QMON_T_CLOSE =>, QMAN_AUT =>, QREMOTE =>, QSIM =>, QLOCK =>, QERR =>, QERR_EXT =>, QwAlarm =>)
   END_RUNG
   RUNG wire#powerrail
      I_Contact( "AV-33.04" )
   END_RUNG wire#w1
   // the same network as SCL:
   #"AV-33.04"(LOCK := #lock,   // "Valve"
               LIOP_SEL := #Init,
               L_AUT := #Init,
               L_REMOTE := #Init,
               L_RESET := #Reset,
               FB_OPEN := "AV-33.04",
               FB_CLOSE := NOT "AV-33.04",
               L_MON := #Init,
               INSTANCE := 'AV-33.04',
               QCMD_OP => "AV-33.04");
END_REGION

REGION Network 40: AV-33.05
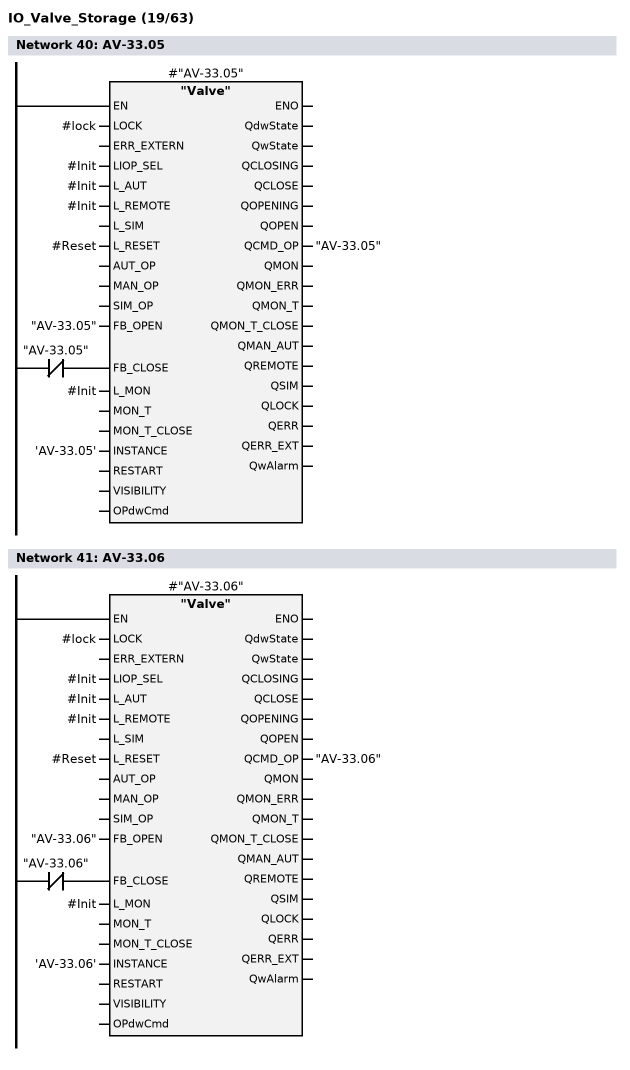
   RUNG wire#powerrail
      #"AV-33.05"(FB_CLOSE := wire#w1, LOCK := #lock, ERR_EXTERN :=, LIOP_SEL := #Init, L_AUT := #Init, L_REMOTE := #Init, L_SIM :=, L_RESET := #Reset, AUT_OP :=, MAN_OP :=, SIM_OP :=, FB_OPEN := "AV-33.05", L_MON := #Init, MON_T :=, MON_T_CLOSE :=, INSTANCE := 'AV-33.05', RESTART :=, VISIBILITY :=, OPdwCmd :=, QdwState =>, QwState =>, QCLOSING =>, QCLOSE =>, QOPENING =>, QOPEN =>, QCMD_OP => "AV-33.05", QMON =>, QMON_ERR =>, QMON_T =>, QMON_T_CLOSE =>, QMAN_AUT =>, QREMOTE =>, QSIM =>, QLOCK =>, QERR =>, QERR_EXT =>, QwAlarm =>)
   END_RUNG
   RUNG wire#powerrail
      I_Contact( "AV-33.05" )
   END_RUNG wire#w1
   // the same network as SCL:
   #"AV-33.05"(LOCK := #lock,   // "Valve"
               LIOP_SEL := #Init,
               L_AUT := #Init,
               L_REMOTE := #Init,
               L_RESET := #Reset,
               FB_OPEN := "AV-33.05",
               FB_CLOSE := NOT "AV-33.05",
               L_MON := #Init,
               INSTANCE := 'AV-33.05',
               QCMD_OP => "AV-33.05");
END_REGION

REGION Network 41: AV-33.06
   RUNG wire#powerrail
      #"AV-33.06"(FB_CLOSE := wire#w1, LOCK := #lock, ERR_EXTERN :=, LIOP_SEL := #Init, L_AUT := #Init, L_REMOTE := #Init, L_SIM :=, L_RESET := #Reset, AUT_OP :=, MAN_OP :=, SIM_OP :=, FB_OPEN := "AV-33.06", L_MON := #Init, MON_T :=, MON_T_CLOSE :=, INSTANCE := 'AV-33.06', RESTART :=, VISIBILITY :=, OPdwCmd :=, QdwState =>, QwState =>, QCLOSING =>, QCLOSE =>, QOPENING =>, QOPEN =>, QCMD_OP => "AV-33.06", QMON =>, QMON_ERR =>, QMON_T =>, QMON_T_CLOSE =>, QMAN_AUT =>, QREMOTE =>, QSIM =>, QLOCK =>, QERR =>, QERR_EXT =>, QwAlarm =>)
   END_RUNG
   RUNG wire#powerrail
      I_Contact( "AV-33.06" )
   END_RUNG wire#w1
   // the same network as SCL:
   #"AV-33.06"(LOCK := #lock,   // "Valve"
               LIOP_SEL := #Init,
               L_AUT := #Init,
               L_REMOTE := #Init,
               L_RESET := #Reset,
               FB_OPEN := "AV-33.06",
               FB_CLOSE := NOT "AV-33.06",
               L_MON := #Init,
               INSTANCE := 'AV-33.06',
               QCMD_OP => "AV-33.06");
END_REGION

REGION Network 42: AV-33.07
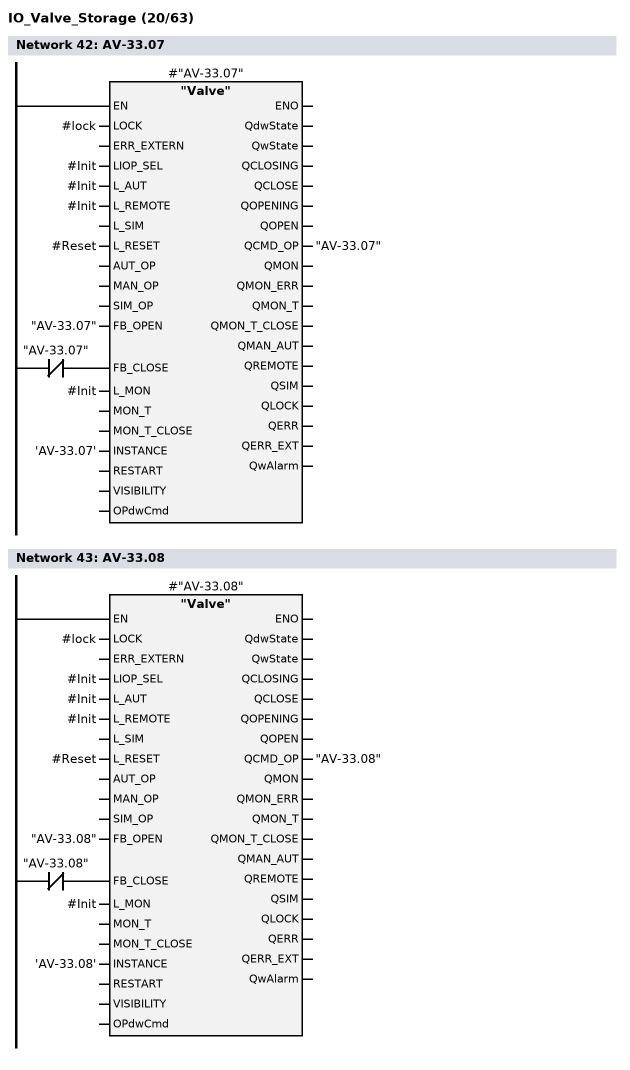
   RUNG wire#powerrail
      #"AV-33.07"(FB_CLOSE := wire#w1, LOCK := #lock, ERR_EXTERN :=, LIOP_SEL := #Init, L_AUT := #Init, L_REMOTE := #Init, L_SIM :=, L_RESET := #Reset, AUT_OP :=, MAN_OP :=, SIM_OP :=, FB_OPEN := "AV-33.07", L_MON := #Init, MON_T :=, MON_T_CLOSE :=, INSTANCE := 'AV-33.07', RESTART :=, VISIBILITY :=, OPdwCmd :=, QdwState =>, QwState =>, QCLOSING =>, QCLOSE =>, QOPENING =>, QOPEN =>, QCMD_OP => "AV-33.07", QMON =>, QMON_ERR =>, QMON_T =>, QMON_T_CLOSE =>, QMAN_AUT =>, QREMOTE =>, QSIM =>, QLOCK =>, QERR =>, QERR_EXT =>, QwAlarm =>)
   END_RUNG
   RUNG wire#powerrail
      I_Contact( "AV-33.07" )
   END_RUNG wire#w1
   // the same network as SCL:
   #"AV-33.07"(LOCK := #lock,   // "Valve"
               LIOP_SEL := #Init,
               L_AUT := #Init,
               L_REMOTE := #Init,
               L_RESET := #Reset,
               FB_OPEN := "AV-33.07",
               FB_CLOSE := NOT "AV-33.07",
               L_MON := #Init,
               INSTANCE := 'AV-33.07',
               QCMD_OP => "AV-33.07");
END_REGION

REGION Network 43: AV-33.08
   RUNG wire#powerrail
      #"AV-33.08"(FB_CLOSE := wire#w1, LOCK := #lock, ERR_EXTERN :=, LIOP_SEL := #Init, L_AUT := #Init, L_REMOTE := #Init, L_SIM :=, L_RESET := #Reset, AUT_OP :=, MAN_OP :=, SIM_OP :=, FB_OPEN := "AV-33.08", L_MON := #Init, MON_T :=, MON_T_CLOSE :=, INSTANCE := 'AV-33.08', RESTART :=, VISIBILITY :=, OPdwCmd :=, QdwState =>, QwState =>, QCLOSING =>, QCLOSE =>, QOPENING =>, QOPEN =>, QCMD_OP => "AV-33.08", QMON =>, QMON_ERR =>, QMON_T =>, QMON_T_CLOSE =>, QMAN_AUT =>, QREMOTE =>, QSIM =>, QLOCK =>, QERR =>, QERR_EXT =>, QwAlarm =>)
   END_RUNG
   RUNG wire#powerrail
      I_Contact( "AV-33.08" )
   END_RUNG wire#w1
   // the same network as SCL:
   #"AV-33.08"(LOCK := #lock,   // "Valve"
               LIOP_SEL := #Init,
               L_AUT := #Init,
               L_REMOTE := #Init,
               L_RESET := #Reset,
               FB_OPEN := "AV-33.08",
               FB_CLOSE := NOT "AV-33.08",
               L_MON := #Init,
               INSTANCE := 'AV-33.08',
               QCMD_OP => "AV-33.08");
END_REGION

REGION Network 44: AV-33.09
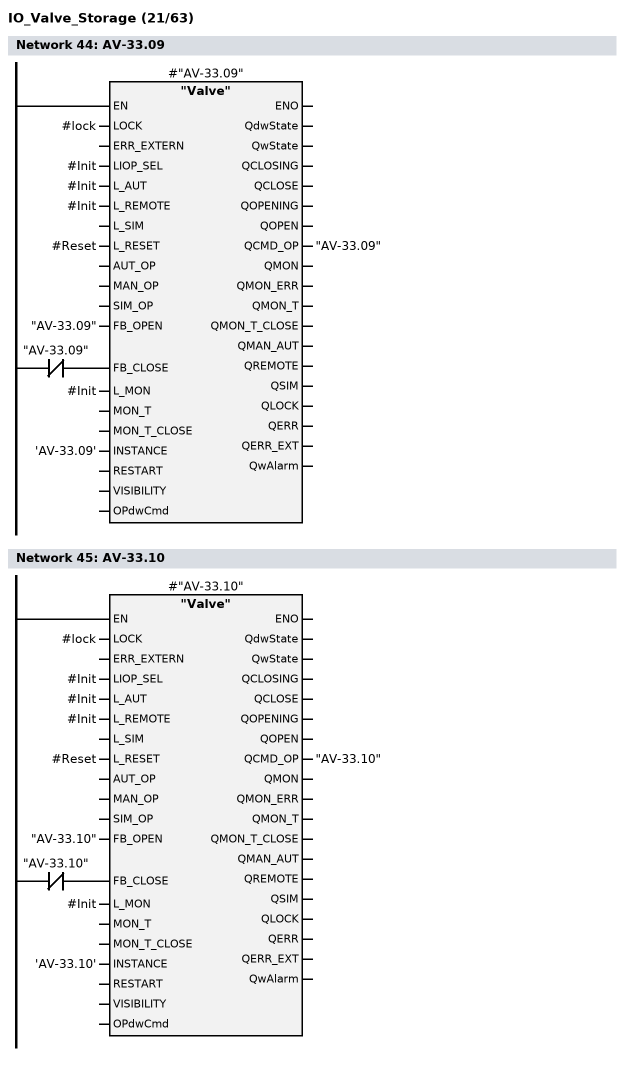
   RUNG wire#powerrail
      #"AV-33.09"(FB_CLOSE := wire#w1, LOCK := #lock, ERR_EXTERN :=, LIOP_SEL := #Init, L_AUT := #Init, L_REMOTE := #Init, L_SIM :=, L_RESET := #Reset, AUT_OP :=, MAN_OP :=, SIM_OP :=, FB_OPEN := "AV-33.09", L_MON := #Init, MON_T :=, MON_T_CLOSE :=, INSTANCE := 'AV-33.09', RESTART :=, VISIBILITY :=, OPdwCmd :=, QdwState =>, QwState =>, QCLOSING =>, QCLOSE =>, QOPENING =>, QOPEN =>, QCMD_OP => "AV-33.09", QMON =>, QMON_ERR =>, QMON_T =>, QMON_T_CLOSE =>, QMAN_AUT =>, QREMOTE =>, QSIM =>, QLOCK =>, QERR =>, QERR_EXT =>, QwAlarm =>)
   END_RUNG
   RUNG wire#powerrail
      I_Contact( "AV-33.09" )
   END_RUNG wire#w1
   // the same network as SCL:
   #"AV-33.09"(LOCK := #lock,   // "Valve"
               LIOP_SEL := #Init,
               L_AUT := #Init,
               L_REMOTE := #Init,
               L_RESET := #Reset,
               FB_OPEN := "AV-33.09",
               FB_CLOSE := NOT "AV-33.09",
               L_MON := #Init,
               INSTANCE := 'AV-33.09',
               QCMD_OP => "AV-33.09");
END_REGION

REGION Network 45: AV-33.10
   RUNG wire#powerrail
      #"AV-33.10"(FB_CLOSE := wire#w1, LOCK := #lock, ERR_EXTERN :=, LIOP_SEL := #Init, L_AUT := #Init, L_REMOTE := #Init, L_SIM :=, L_RESET := #Reset, AUT_OP :=, MAN_OP :=, SIM_OP :=, FB_OPEN := "AV-33.10", L_MON := #Init, MON_T :=, MON_T_CLOSE :=, INSTANCE := 'AV-33.10', RESTART :=, VISIBILITY :=, OPdwCmd :=, QdwState =>, QwState =>, QCLOSING =>, QCLOSE =>, QOPENING =>, QOPEN =>, QCMD_OP => "AV-33.10", QMON =>, QMON_ERR =>, QMON_T =>, QMON_T_CLOSE =>, QMAN_AUT =>, QREMOTE =>, QSIM =>, QLOCK =>, QERR =>, QERR_EXT =>, QwAlarm =>)
   END_RUNG
   RUNG wire#powerrail
      I_Contact( "AV-33.10" )
   END_RUNG wire#w1
   // the same network as SCL:
   #"AV-33.10"(LOCK := #lock,   // "Valve"
               LIOP_SEL := #Init,
               L_AUT := #Init,
               L_REMOTE := #Init,
               L_RESET := #Reset,
               FB_OPEN := "AV-33.10",
               FB_CLOSE := NOT "AV-33.10",
               L_MON := #Init,
               INSTANCE := 'AV-33.10',
               QCMD_OP => "AV-33.10");
END_REGION

REGION Network 46: AV-33.11
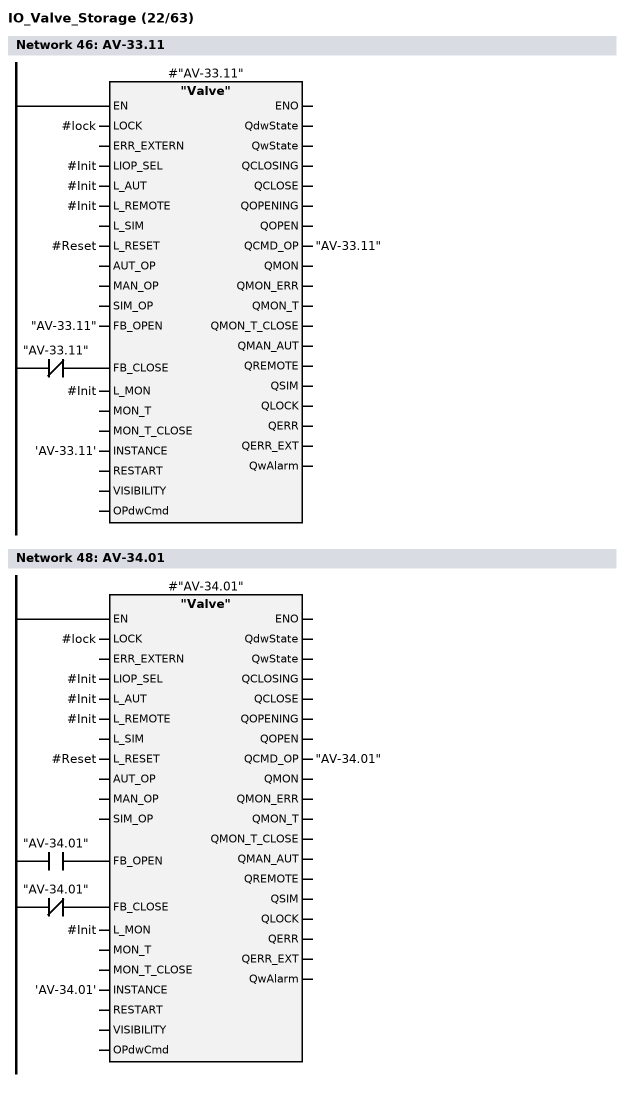
   RUNG wire#powerrail
      #"AV-33.11"(FB_CLOSE := wire#w1, LOCK := #lock, ERR_EXTERN :=, LIOP_SEL := #Init, L_AUT := #Init, L_REMOTE := #Init, L_SIM :=, L_RESET := #Reset, AUT_OP :=, MAN_OP :=, SIM_OP :=, FB_OPEN := "AV-33.11", L_MON := #Init, MON_T :=, MON_T_CLOSE :=, INSTANCE := 'AV-33.11', RESTART :=, VISIBILITY :=, OPdwCmd :=, QdwState =>, QwState =>, QCLOSING =>, QCLOSE =>, QOPENING =>, QOPEN =>, QCMD_OP => "AV-33.11", QMON =>, QMON_ERR =>, QMON_T =>, QMON_T_CLOSE =>, QMAN_AUT =>, QREMOTE =>, QSIM =>, QLOCK =>, QERR =>, QERR_EXT =>, QwAlarm =>)
   END_RUNG
   RUNG wire#powerrail
      I_Contact( "AV-33.11" )
   END_RUNG wire#w1
   // the same network as SCL:
   #"AV-33.11"(LOCK := #lock,   // "Valve"
               LIOP_SEL := #Init,
               L_AUT := #Init,
               L_REMOTE := #Init,
               L_RESET := #Reset,
               FB_OPEN := "AV-33.11",
               FB_CLOSE := NOT "AV-33.11",
               L_MON := #Init,
               INSTANCE := 'AV-33.11',
               QCMD_OP => "AV-33.11");
END_REGION

REGION Network 48: AV-34.01
   RUNG wire#powerrail
      #"AV-34.01"(FB_OPEN := wire#w1, FB_CLOSE := wire#w2, LOCK := #lock, ERR_EXTERN :=, LIOP_SEL := #Init, L_AUT := #Init, L_REMOTE := #Init, L_SIM :=, L_RESET := #Reset, AUT_OP :=, MAN_OP :=, SIM_OP :=, L_MON := #Init, MON_T :=, MON_T_CLOSE :=, INSTANCE := 'AV-34.01', RESTART :=, VISIBILITY :=, OPdwCmd :=, QdwState =>, QwState =>, QCLOSING =>, QCLOSE =>, QOPENING =>, QOPEN =>, QCMD_OP => "AV-34.01", QMON =>, QMON_ERR =>, QMON_T =>, QMON_T_CLOSE =>, QMAN_AUT =>, QREMOTE =>, QSIM =>, QLOCK =>, QERR =>, QERR_EXT =>, QwAlarm =>)
   END_RUNG
   RUNG wire#powerrail
      Contact( "AV-34.01" )
   END_RUNG wire#w1
   RUNG wire#powerrail
      I_Contact( "AV-34.01" )
   END_RUNG wire#w2
   // the same network as SCL:
   #"AV-34.01"(LOCK := #lock,   // "Valve"
               LIOP_SEL := #Init,
               L_AUT := #Init,
               L_REMOTE := #Init,
               L_RESET := #Reset,
               FB_OPEN := "AV-34.01",
               FB_CLOSE := NOT "AV-34.01",
               L_MON := #Init,
               INSTANCE := 'AV-34.01',
               QCMD_OP => "AV-34.01");
END_REGION

REGION Network 49: AV-34.02
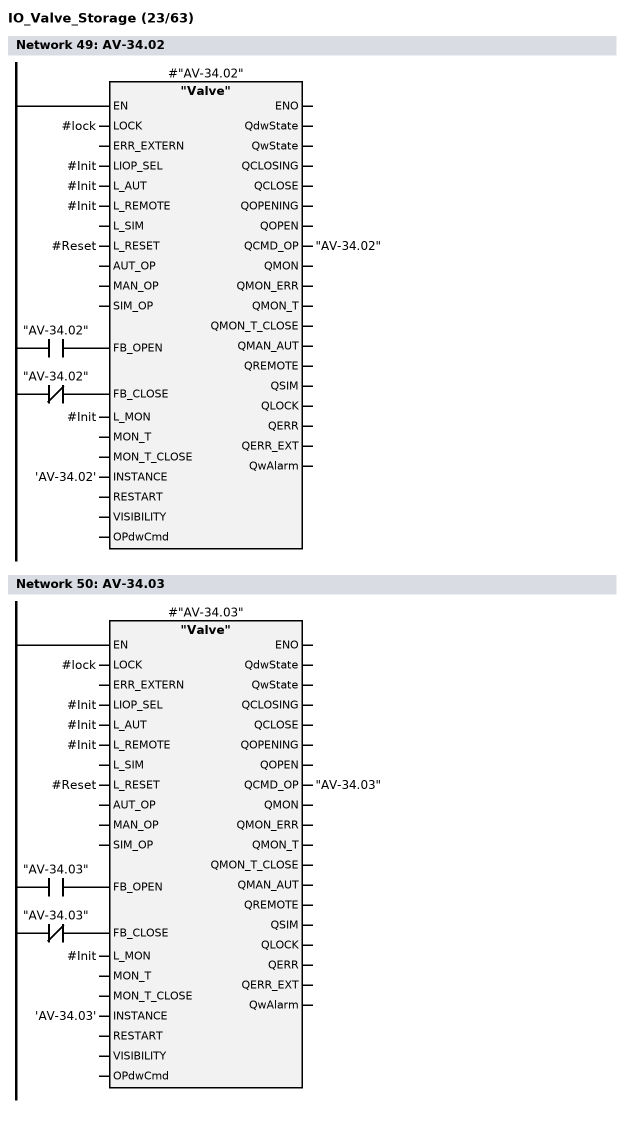
   RUNG wire#powerrail
      #"AV-34.02"(FB_OPEN := wire#w1, FB_CLOSE := wire#w2, LOCK := #lock, ERR_EXTERN :=, LIOP_SEL := #Init, L_AUT := #Init, L_REMOTE := #Init, L_SIM :=, L_RESET := #Reset, AUT_OP :=, MAN_OP :=, SIM_OP :=, L_MON := #Init, MON_T :=, MON_T_CLOSE :=, INSTANCE := 'AV-34.02', RESTART :=, VISIBILITY :=, OPdwCmd :=, QdwState =>, QwState =>, QCLOSING =>, QCLOSE =>, QOPENING =>, QOPEN =>, QCMD_OP => "AV-34.02", QMON =>, QMON_ERR =>, QMON_T =>, QMON_T_CLOSE =>, QMAN_AUT =>, QREMOTE =>, QSIM =>, QLOCK =>, QERR =>, QERR_EXT =>, QwAlarm =>)
   END_RUNG
   RUNG wire#powerrail
      Contact( "AV-34.02" )
   END_RUNG wire#w1
   RUNG wire#powerrail
      I_Contact( "AV-34.02" )
   END_RUNG wire#w2
   // the same network as SCL:
   #"AV-34.02"(LOCK := #lock,   // "Valve"
               LIOP_SEL := #Init,
               L_AUT := #Init,
               L_REMOTE := #Init,
               L_RESET := #Reset,
               FB_OPEN := "AV-34.02",
               FB_CLOSE := NOT "AV-34.02",
               L_MON := #Init,
               INSTANCE := 'AV-34.02',
               QCMD_OP => "AV-34.02");
END_REGION

REGION Network 50: AV-34.03
   RUNG wire#powerrail
      #"AV-34.03"(FB_OPEN := wire#w1, FB_CLOSE := wire#w2, LOCK := #lock, ERR_EXTERN :=, LIOP_SEL := #Init, L_AUT := #Init, L_REMOTE := #Init, L_SIM :=, L_RESET := #Reset, AUT_OP :=, MAN_OP :=, SIM_OP :=, L_MON := #Init, MON_T :=, MON_T_CLOSE :=, INSTANCE := 'AV-34.03', RESTART :=, VISIBILITY :=, OPdwCmd :=, QdwState =>, QwState =>, QCLOSING =>, QCLOSE =>, QOPENING =>, QOPEN =>, QCMD_OP => "AV-34.03", QMON =>, QMON_ERR =>, QMON_T =>, QMON_T_CLOSE =>, QMAN_AUT =>, QREMOTE =>, QSIM =>, QLOCK =>, QERR =>, QERR_EXT =>, QwAlarm =>)
   END_RUNG
   RUNG wire#powerrail
      Contact( "AV-34.03" )
   END_RUNG wire#w1
   RUNG wire#powerrail
      I_Contact( "AV-34.03" )
   END_RUNG wire#w2
   // the same network as SCL:
   #"AV-34.03"(LOCK := #lock,   // "Valve"
               LIOP_SEL := #Init,
               L_AUT := #Init,
               L_REMOTE := #Init,
               L_RESET := #Reset,
               FB_OPEN := "AV-34.03",
               FB_CLOSE := NOT "AV-34.03",
               L_MON := #Init,
               INSTANCE := 'AV-34.03',
               QCMD_OP => "AV-34.03");
END_REGION

REGION Network 51: AV-34.04
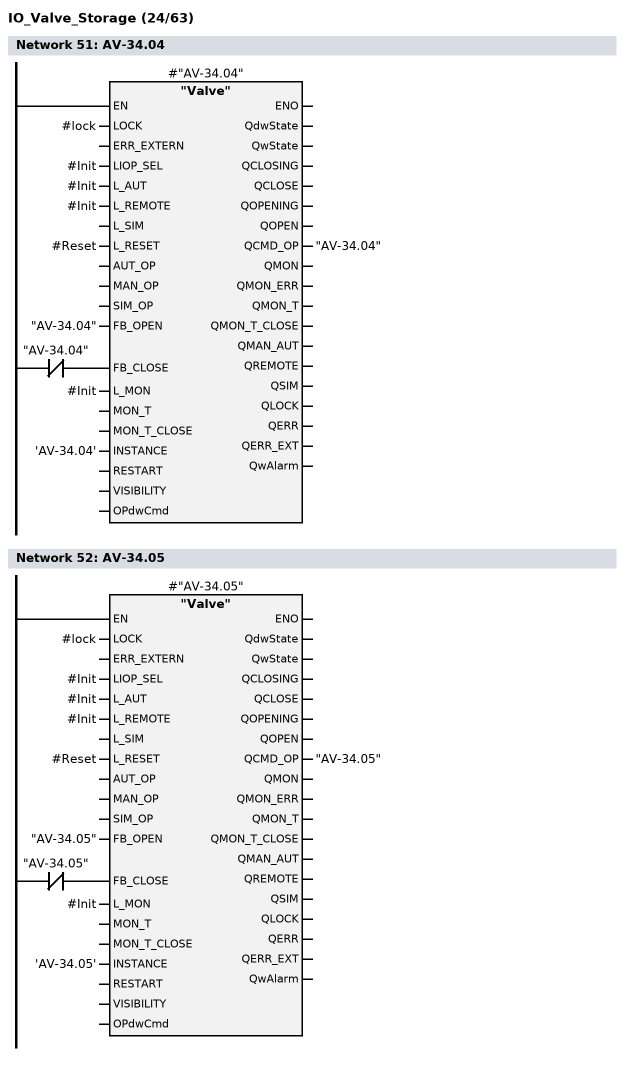
   RUNG wire#powerrail
      #"AV-34.04"(FB_CLOSE := wire#w1, LOCK := #lock, ERR_EXTERN :=, LIOP_SEL := #Init, L_AUT := #Init, L_REMOTE := #Init, L_SIM :=, L_RESET := #Reset, AUT_OP :=, MAN_OP :=, SIM_OP :=, FB_OPEN := "AV-34.04", L_MON := #Init, MON_T :=, MON_T_CLOSE :=, INSTANCE := 'AV-34.04', RESTART :=, VISIBILITY :=, OPdwCmd :=, QdwState =>, QwState =>, QCLOSING =>, QCLOSE =>, QOPENING =>, QOPEN =>, QCMD_OP => "AV-34.04", QMON =>, QMON_ERR =>, QMON_T =>, QMON_T_CLOSE =>, QMAN_AUT =>, QREMOTE =>, QSIM =>, QLOCK =>, QERR =>, QERR_EXT =>, QwAlarm =>)
   END_RUNG
   RUNG wire#powerrail
      I_Contact( "AV-34.04" )
   END_RUNG wire#w1
   // the same network as SCL:
   #"AV-34.04"(LOCK := #lock,   // "Valve"
               LIOP_SEL := #Init,
               L_AUT := #Init,
               L_REMOTE := #Init,
               L_RESET := #Reset,
               FB_OPEN := "AV-34.04",
               FB_CLOSE := NOT "AV-34.04",
               L_MON := #Init,
               INSTANCE := 'AV-34.04',
               QCMD_OP => "AV-34.04");
END_REGION

REGION Network 52: AV-34.05
   RUNG wire#powerrail
      #"AV-34.05"(FB_CLOSE := wire#w1, LOCK := #lock, ERR_EXTERN :=, LIOP_SEL := #Init, L_AUT := #Init, L_REMOTE := #Init, L_SIM :=, L_RESET := #Reset, AUT_OP :=, MAN_OP :=, SIM_OP :=, FB_OPEN := "AV-34.05", L_MON := #Init, MON_T :=, MON_T_CLOSE :=, INSTANCE := 'AV-34.05', RESTART :=, VISIBILITY :=, OPdwCmd :=, QdwState =>, QwState =>, QCLOSING =>, QCLOSE =>, QOPENING =>, QOPEN =>, QCMD_OP => "AV-34.05", QMON =>, QMON_ERR =>, QMON_T =>, QMON_T_CLOSE =>, QMAN_AUT =>, QREMOTE =>, QSIM =>, QLOCK =>, QERR =>, QERR_EXT =>, QwAlarm =>)
   END_RUNG
   RUNG wire#powerrail
      I_Contact( "AV-34.05" )
   END_RUNG wire#w1
   // the same network as SCL:
   #"AV-34.05"(LOCK := #lock,   // "Valve"
               LIOP_SEL := #Init,
               L_AUT := #Init,
               L_REMOTE := #Init,
               L_RESET := #Reset,
               FB_OPEN := "AV-34.05",
               FB_CLOSE := NOT "AV-34.05",
               L_MON := #Init,
               INSTANCE := 'AV-34.05',
               QCMD_OP => "AV-34.05");
END_REGION

REGION Network 53: AV-34.06
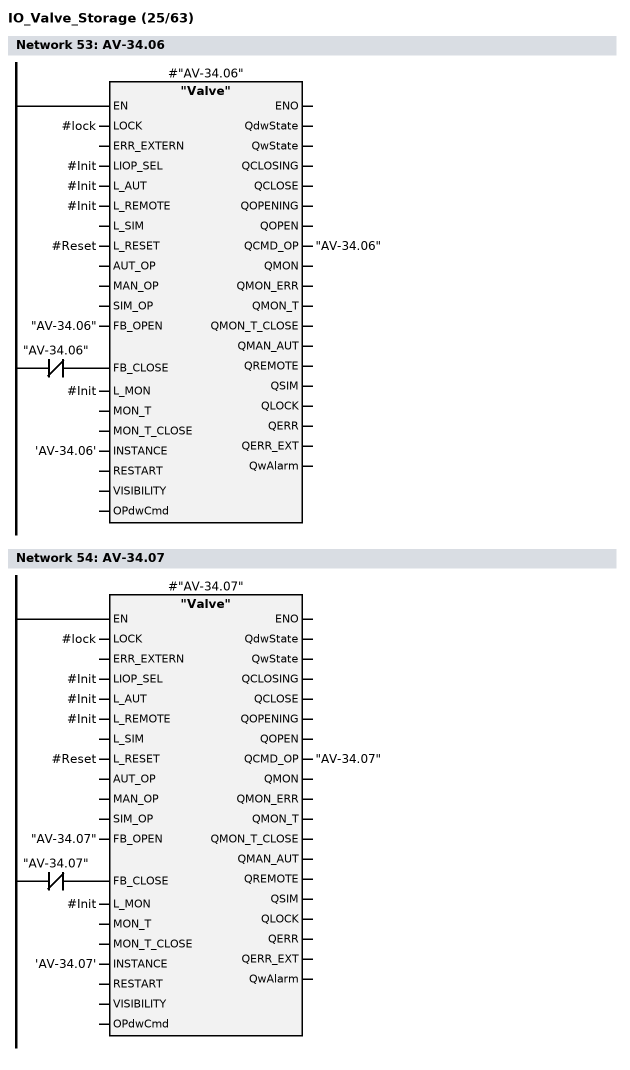
   RUNG wire#powerrail
      #"AV-34.06"(FB_CLOSE := wire#w1, LOCK := #lock, ERR_EXTERN :=, LIOP_SEL := #Init, L_AUT := #Init, L_REMOTE := #Init, L_SIM :=, L_RESET := #Reset, AUT_OP :=, MAN_OP :=, SIM_OP :=, FB_OPEN := "AV-34.06", L_MON := #Init, MON_T :=, MON_T_CLOSE :=, INSTANCE := 'AV-34.06', RESTART :=, VISIBILITY :=, OPdwCmd :=, QdwState =>, QwState =>, QCLOSING =>, QCLOSE =>, QOPENING =>, QOPEN =>, QCMD_OP => "AV-34.06", QMON =>, QMON_ERR =>, QMON_T =>, QMON_T_CLOSE =>, QMAN_AUT =>, QREMOTE =>, QSIM =>, QLOCK =>, QERR =>, QERR_EXT =>, QwAlarm =>)
   END_RUNG
   RUNG wire#powerrail
      I_Contact( "AV-34.06" )
   END_RUNG wire#w1
   // the same network as SCL:
   #"AV-34.06"(LOCK := #lock,   // "Valve"
               LIOP_SEL := #Init,
               L_AUT := #Init,
               L_REMOTE := #Init,
               L_RESET := #Reset,
               FB_OPEN := "AV-34.06",
               FB_CLOSE := NOT "AV-34.06",
               L_MON := #Init,
               INSTANCE := 'AV-34.06',
               QCMD_OP => "AV-34.06");
END_REGION

REGION Network 54: AV-34.07
   RUNG wire#powerrail
      #"AV-34.07"(FB_CLOSE := wire#w1, LOCK := #lock, ERR_EXTERN :=, LIOP_SEL := #Init, L_AUT := #Init, L_REMOTE := #Init, L_SIM :=, L_RESET := #Reset, AUT_OP :=, MAN_OP :=, SIM_OP :=, FB_OPEN := "AV-34.07", L_MON := #Init, MON_T :=, MON_T_CLOSE :=, INSTANCE := 'AV-34.07', RESTART :=, VISIBILITY :=, OPdwCmd :=, QdwState =>, QwState =>, QCLOSING =>, QCLOSE =>, QOPENING =>, QOPEN =>, QCMD_OP => "AV-34.07", QMON =>, QMON_ERR =>, QMON_T =>, QMON_T_CLOSE =>, QMAN_AUT =>, QREMOTE =>, QSIM =>, QLOCK =>, QERR =>, QERR_EXT =>, QwAlarm =>)
   END_RUNG
   RUNG wire#powerrail
      I_Contact( "AV-34.07" )
   END_RUNG wire#w1
   // the same network as SCL:
   #"AV-34.07"(LOCK := #lock,   // "Valve"
               LIOP_SEL := #Init,
               L_AUT := #Init,
               L_REMOTE := #Init,
               L_RESET := #Reset,
               FB_OPEN := "AV-34.07",
               FB_CLOSE := NOT "AV-34.07",
               L_MON := #Init,
               INSTANCE := 'AV-34.07',
               QCMD_OP => "AV-34.07");
END_REGION

REGION Network 55: AV-34.08
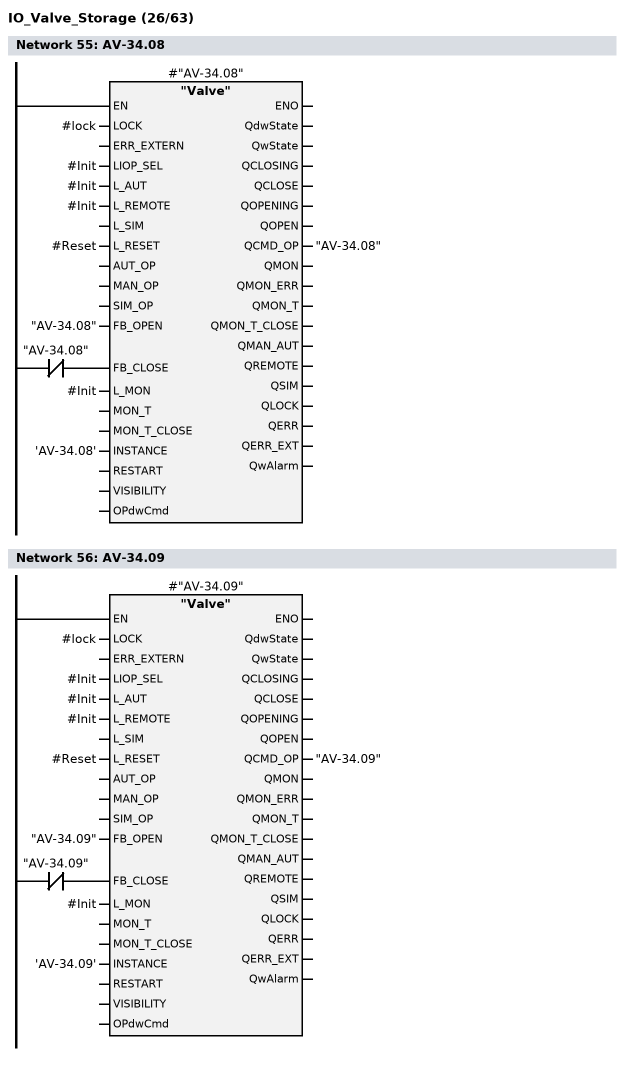
   RUNG wire#powerrail
      #"AV-34.08"(FB_CLOSE := wire#w1, LOCK := #lock, ERR_EXTERN :=, LIOP_SEL := #Init, L_AUT := #Init, L_REMOTE := #Init, L_SIM :=, L_RESET := #Reset, AUT_OP :=, MAN_OP :=, SIM_OP :=, FB_OPEN := "AV-34.08", L_MON := #Init, MON_T :=, MON_T_CLOSE :=, INSTANCE := 'AV-34.08', RESTART :=, VISIBILITY :=, OPdwCmd :=, QdwState =>, QwState =>, QCLOSING =>, QCLOSE =>, QOPENING =>, QOPEN =>, QCMD_OP => "AV-34.08", QMON =>, QMON_ERR =>, QMON_T =>, QMON_T_CLOSE =>, QMAN_AUT =>, QREMOTE =>, QSIM =>, QLOCK =>, QERR =>, QERR_EXT =>, QwAlarm =>)
   END_RUNG
   RUNG wire#powerrail
      I_Contact( "AV-34.08" )
   END_RUNG wire#w1
   // the same network as SCL:
   #"AV-34.08"(LOCK := #lock,   // "Valve"
               LIOP_SEL := #Init,
               L_AUT := #Init,
               L_REMOTE := #Init,
               L_RESET := #Reset,
               FB_OPEN := "AV-34.08",
               FB_CLOSE := NOT "AV-34.08",
               L_MON := #Init,
               INSTANCE := 'AV-34.08',
               QCMD_OP => "AV-34.08");
END_REGION

REGION Network 56: AV-34.09
   RUNG wire#powerrail
      #"AV-34.09"(FB_CLOSE := wire#w1, LOCK := #lock, ERR_EXTERN :=, LIOP_SEL := #Init, L_AUT := #Init, L_REMOTE := #Init, L_SIM :=, L_RESET := #Reset, AUT_OP :=, MAN_OP :=, SIM_OP :=, FB_OPEN := "AV-34.09", L_MON := #Init, MON_T :=, MON_T_CLOSE :=, INSTANCE := 'AV-34.09', RESTART :=, VISIBILITY :=, OPdwCmd :=, QdwState =>, QwState =>, QCLOSING =>, QCLOSE =>, QOPENING =>, QOPEN =>, QCMD_OP => "AV-34.09", QMON =>, QMON_ERR =>, QMON_T =>, QMON_T_CLOSE =>, QMAN_AUT =>, QREMOTE =>, QSIM =>, QLOCK =>, QERR =>, QERR_EXT =>, QwAlarm =>)
   END_RUNG
   RUNG wire#powerrail
      I_Contact( "AV-34.09" )
   END_RUNG wire#w1
   // the same network as SCL:
   #"AV-34.09"(LOCK := #lock,   // "Valve"
               LIOP_SEL := #Init,
               L_AUT := #Init,
               L_REMOTE := #Init,
               L_RESET := #Reset,
               FB_OPEN := "AV-34.09",
               FB_CLOSE := NOT "AV-34.09",
               L_MON := #Init,
               INSTANCE := 'AV-34.09',
               QCMD_OP => "AV-34.09");
END_REGION

REGION Network 57: AV-34.10
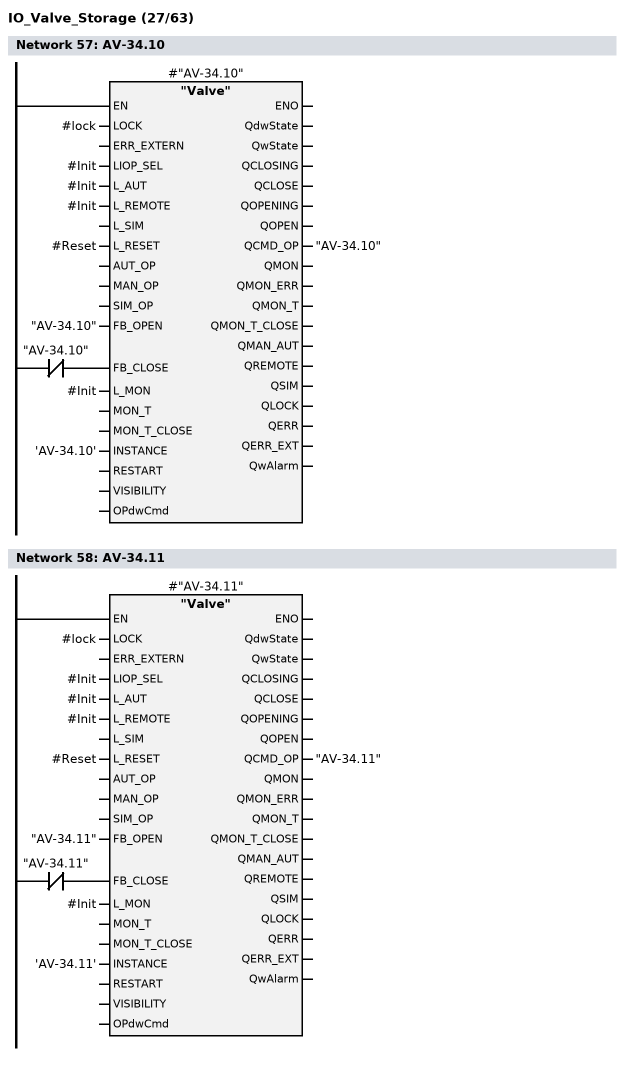
   RUNG wire#powerrail
      #"AV-34.10"(FB_CLOSE := wire#w1, LOCK := #lock, ERR_EXTERN :=, LIOP_SEL := #Init, L_AUT := #Init, L_REMOTE := #Init, L_SIM :=, L_RESET := #Reset, AUT_OP :=, MAN_OP :=, SIM_OP :=, FB_OPEN := "AV-34.10", L_MON := #Init, MON_T :=, MON_T_CLOSE :=, INSTANCE := 'AV-34.10', RESTART :=, VISIBILITY :=, OPdwCmd :=, QdwState =>, QwState =>, QCLOSING =>, QCLOSE =>, QOPENING =>, QOPEN =>, QCMD_OP => "AV-34.10", QMON =>, QMON_ERR =>, QMON_T =>, QMON_T_CLOSE =>, QMAN_AUT =>, QREMOTE =>, QSIM =>, QLOCK =>, QERR =>, QERR_EXT =>, QwAlarm =>)
   END_RUNG
   RUNG wire#powerrail
      I_Contact( "AV-34.10" )
   END_RUNG wire#w1
   // the same network as SCL:
   #"AV-34.10"(LOCK := #lock,   // "Valve"
               LIOP_SEL := #Init,
               L_AUT := #Init,
               L_REMOTE := #Init,
               L_RESET := #Reset,
               FB_OPEN := "AV-34.10",
               FB_CLOSE := NOT "AV-34.10",
               L_MON := #Init,
               INSTANCE := 'AV-34.10',
               QCMD_OP => "AV-34.10");
END_REGION

REGION Network 58: AV-34.11
   RUNG wire#powerrail
      #"AV-34.11"(FB_CLOSE := wire#w1, LOCK := #lock, ERR_EXTERN :=, LIOP_SEL := #Init, L_AUT := #Init, L_REMOTE := #Init, L_SIM :=, L_RESET := #Reset, AUT_OP :=, MAN_OP :=, SIM_OP :=, FB_OPEN := "AV-34.11", L_MON := #Init, MON_T :=, MON_T_CLOSE :=, INSTANCE := 'AV-34.11', RESTART :=, VISIBILITY :=, OPdwCmd :=, QdwState =>, QwState =>, QCLOSING =>, QCLOSE =>, QOPENING =>, QOPEN =>, QCMD_OP => "AV-34.11", QMON =>, QMON_ERR =>, QMON_T =>, QMON_T_CLOSE =>, QMAN_AUT =>, QREMOTE =>, QSIM =>, QLOCK =>, QERR =>, QERR_EXT =>, QwAlarm =>)
   END_RUNG
   RUNG wire#powerrail
      I_Contact( "AV-34.11" )
   END_RUNG wire#w1
   // the same network as SCL:
   #"AV-34.11"(LOCK := #lock,   // "Valve"
               LIOP_SEL := #Init,
               L_AUT := #Init,
               L_REMOTE := #Init,
               L_RESET := #Reset,
               FB_OPEN := "AV-34.11",
               FB_CLOSE := NOT "AV-34.11",
               L_MON := #Init,
               INSTANCE := 'AV-34.11',
               QCMD_OP => "AV-34.11");
END_REGION

REGION Network 59: AV-34.12
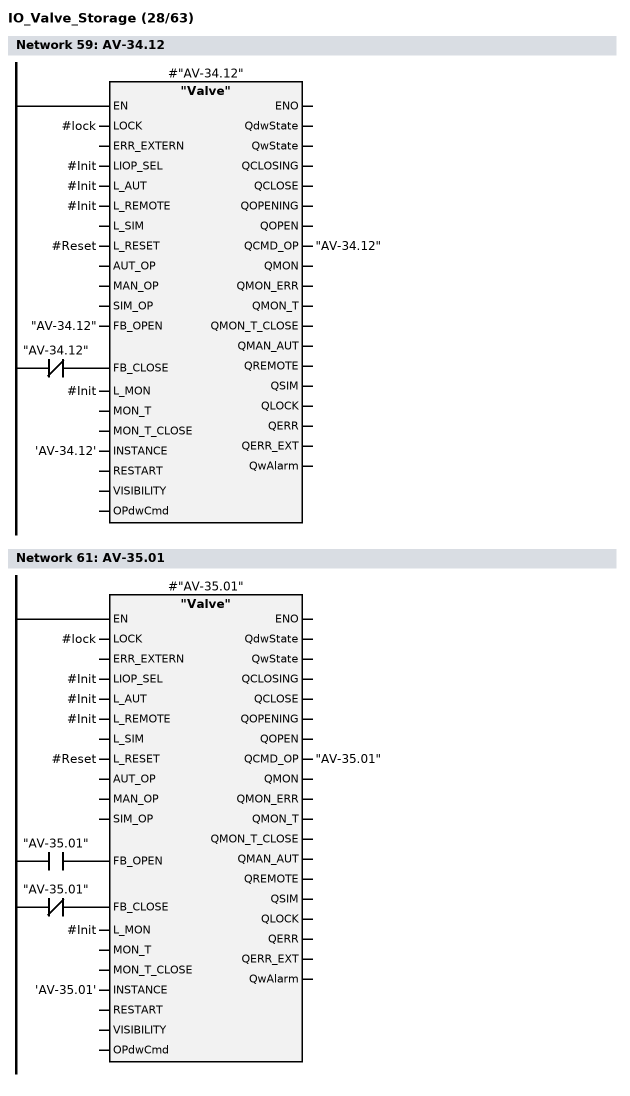
   RUNG wire#powerrail
      #"AV-34.12"(FB_CLOSE := wire#w1, LOCK := #lock, ERR_EXTERN :=, LIOP_SEL := #Init, L_AUT := #Init, L_REMOTE := #Init, L_SIM :=, L_RESET := #Reset, AUT_OP :=, MAN_OP :=, SIM_OP :=, FB_OPEN := "AV-34.12", L_MON := #Init, MON_T :=, MON_T_CLOSE :=, INSTANCE := 'AV-34.12', RESTART :=, VISIBILITY :=, OPdwCmd :=, QdwState =>, QwState =>, QCLOSING =>, QCLOSE =>, QOPENING =>, QOPEN =>, QCMD_OP => "AV-34.12", QMON =>, QMON_ERR =>, QMON_T =>, QMON_T_CLOSE =>, QMAN_AUT =>, QREMOTE =>, QSIM =>, QLOCK =>, QERR =>, QERR_EXT =>, QwAlarm =>)
   END_RUNG
   RUNG wire#powerrail
      I_Contact( "AV-34.12" )
   END_RUNG wire#w1
   // the same network as SCL:
   #"AV-34.12"(LOCK := #lock,   // "Valve"
               LIOP_SEL := #Init,
               L_AUT := #Init,
               L_REMOTE := #Init,
               L_RESET := #Reset,
               FB_OPEN := "AV-34.12",
               FB_CLOSE := NOT "AV-34.12",
               L_MON := #Init,
               INSTANCE := 'AV-34.12',
               QCMD_OP => "AV-34.12");
END_REGION

REGION Network 61: AV-35.01
   RUNG wire#powerrail
      #"AV-35.01"(FB_OPEN := wire#w1, FB_CLOSE := wire#w2, LOCK := #lock, ERR_EXTERN :=, LIOP_SEL := #Init, L_AUT := #Init, L_REMOTE := #Init, L_SIM :=, L_RESET := #Reset, AUT_OP :=, MAN_OP :=, SIM_OP :=, L_MON := #Init, MON_T :=, MON_T_CLOSE :=, INSTANCE := 'AV-35.01', RESTART :=, VISIBILITY :=, OPdwCmd :=, QdwState =>, QwState =>, QCLOSING =>, QCLOSE =>, QOPENING =>, QOPEN =>, QCMD_OP => "AV-35.01", QMON =>, QMON_ERR =>, QMON_T =>, QMON_T_CLOSE =>, QMAN_AUT =>, QREMOTE =>, QSIM =>, QLOCK =>, QERR =>, QERR_EXT =>, QwAlarm =>)
   END_RUNG
   RUNG wire#powerrail
      Contact( "AV-35.01" )
   END_RUNG wire#w1
   RUNG wire#powerrail
      I_Contact( "AV-35.01" )
   END_RUNG wire#w2
   // the same network as SCL:
   #"AV-35.01"(LOCK := #lock,   // "Valve"
               LIOP_SEL := #Init,
               L_AUT := #Init,
               L_REMOTE := #Init,
               L_RESET := #Reset,
               FB_OPEN := "AV-35.01",
               FB_CLOSE := NOT "AV-35.01",
               L_MON := #Init,
               INSTANCE := 'AV-35.01',
               QCMD_OP => "AV-35.01");
END_REGION

REGION Network 62: AV-35.02
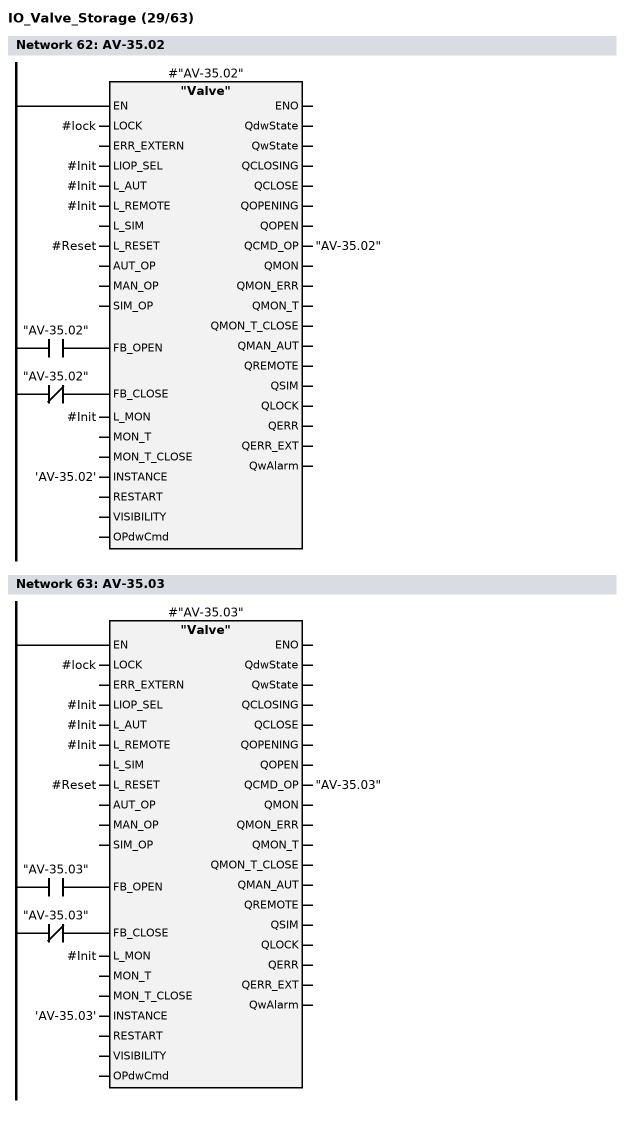
   RUNG wire#powerrail
      #"AV-35.02"(FB_OPEN := wire#w1, FB_CLOSE := wire#w2, LOCK := #lock, ERR_EXTERN :=, LIOP_SEL := #Init, L_AUT := #Init, L_REMOTE := #Init, L_SIM :=, L_RESET := #Reset, AUT_OP :=, MAN_OP :=, SIM_OP :=, L_MON := #Init, MON_T :=, MON_T_CLOSE :=, INSTANCE := 'AV-35.02', RESTART :=, VISIBILITY :=, OPdwCmd :=, QdwState =>, QwState =>, QCLOSING =>, QCLOSE =>, QOPENING =>, QOPEN =>, QCMD_OP => "AV-35.02", QMON =>, QMON_ERR =>, QMON_T =>, QMON_T_CLOSE =>, QMAN_AUT =>, QREMOTE =>, QSIM =>, QLOCK =>, QERR =>, QERR_EXT =>, QwAlarm =>)
   END_RUNG
   RUNG wire#powerrail
      Contact( "AV-35.02" )
   END_RUNG wire#w1
   RUNG wire#powerrail
      I_Contact( "AV-35.02" )
   END_RUNG wire#w2
   // the same network as SCL:
   #"AV-35.02"(LOCK := #lock,   // "Valve"
               LIOP_SEL := #Init,
               L_AUT := #Init,
               L_REMOTE := #Init,
               L_RESET := #Reset,
               FB_OPEN := "AV-35.02",
               FB_CLOSE := NOT "AV-35.02",
               L_MON := #Init,
               INSTANCE := 'AV-35.02',
               QCMD_OP => "AV-35.02");
END_REGION

REGION Network 63: AV-35.03
   RUNG wire#powerrail
      #"AV-35.03"(FB_OPEN := wire#w1, FB_CLOSE := wire#w2, LOCK := #lock, ERR_EXTERN :=, LIOP_SEL := #Init, L_AUT := #Init, L_REMOTE := #Init, L_SIM :=, L_RESET := #Reset, AUT_OP :=, MAN_OP :=, SIM_OP :=, L_MON := #Init, MON_T :=, MON_T_CLOSE :=, INSTANCE := 'AV-35.03', RESTART :=, VISIBILITY :=, OPdwCmd :=, QdwState =>, QwState =>, QCLOSING =>, QCLOSE =>, QOPENING =>, QOPEN =>, QCMD_OP => "AV-35.03", QMON =>, QMON_ERR =>, QMON_T =>, QMON_T_CLOSE =>, QMAN_AUT =>, QREMOTE =>, QSIM =>, QLOCK =>, QERR =>, QERR_EXT =>, QwAlarm =>)
   END_RUNG
   RUNG wire#powerrail
      Contact( "AV-35.03" )
   END_RUNG wire#w1
   RUNG wire#powerrail
      I_Contact( "AV-35.03" )
   END_RUNG wire#w2
   // the same network as SCL:
   #"AV-35.03"(LOCK := #lock,   // "Valve"
               LIOP_SEL := #Init,
               L_AUT := #Init,
               L_REMOTE := #Init,
               L_RESET := #Reset,
               FB_OPEN := "AV-35.03",
               FB_CLOSE := NOT "AV-35.03",
               L_MON := #Init,
               INSTANCE := 'AV-35.03',
               QCMD_OP => "AV-35.03");
END_REGION

REGION Network 64: AV-35.04
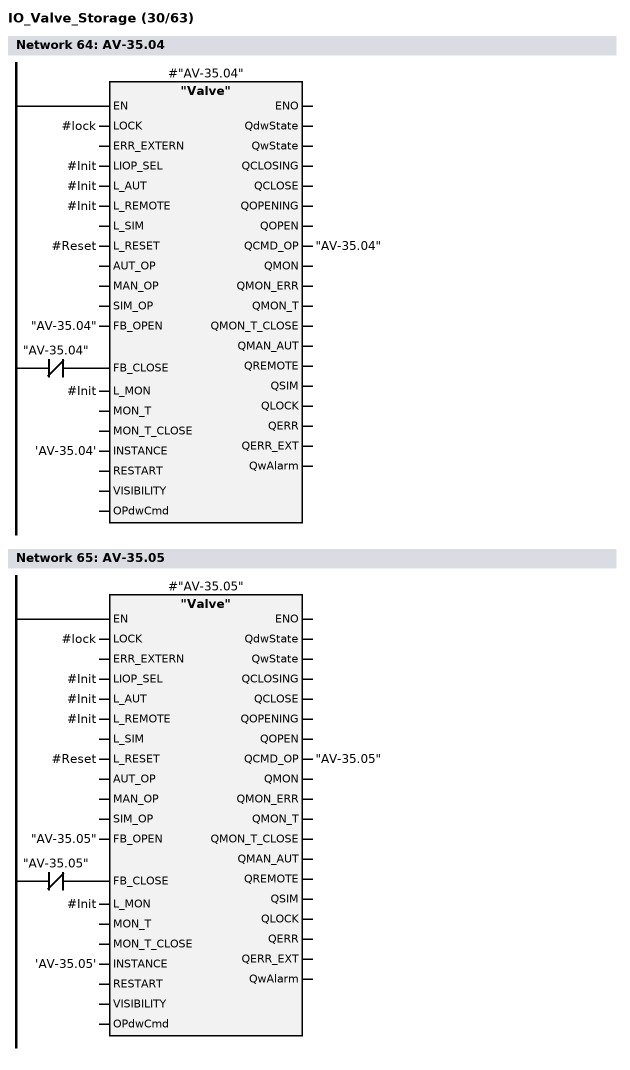
   RUNG wire#powerrail
      #"AV-35.04"(FB_CLOSE := wire#w1, LOCK := #lock, ERR_EXTERN :=, LIOP_SEL := #Init, L_AUT := #Init, L_REMOTE := #Init, L_SIM :=, L_RESET := #Reset, AUT_OP :=, MAN_OP :=, SIM_OP :=, FB_OPEN := "AV-35.04", L_MON := #Init, MON_T :=, MON_T_CLOSE :=, INSTANCE := 'AV-35.04', RESTART :=, VISIBILITY :=, OPdwCmd :=, QdwState =>, QwState =>, QCLOSING =>, QCLOSE =>, QOPENING =>, QOPEN =>, QCMD_OP => "AV-35.04", QMON =>, QMON_ERR =>, QMON_T =>, QMON_T_CLOSE =>, QMAN_AUT =>, QREMOTE =>, QSIM =>, QLOCK =>, QERR =>, QERR_EXT =>, QwAlarm =>)
   END_RUNG
   RUNG wire#powerrail
      I_Contact( "AV-35.04" )
   END_RUNG wire#w1
   // the same network as SCL:
   #"AV-35.04"(LOCK := #lock,   // "Valve"
               LIOP_SEL := #Init,
               L_AUT := #Init,
               L_REMOTE := #Init,
               L_RESET := #Reset,
               FB_OPEN := "AV-35.04",
               FB_CLOSE := NOT "AV-35.04",
               L_MON := #Init,
               INSTANCE := 'AV-35.04',
               QCMD_OP => "AV-35.04");
END_REGION

REGION Network 65: AV-35.05
   RUNG wire#powerrail
      #"AV-35.05"(FB_CLOSE := wire#w1, LOCK := #lock, ERR_EXTERN :=, LIOP_SEL := #Init, L_AUT := #Init, L_REMOTE := #Init, L_SIM :=, L_RESET := #Reset, AUT_OP :=, MAN_OP :=, SIM_OP :=, FB_OPEN := "AV-35.05", L_MON := #Init, MON_T :=, MON_T_CLOSE :=, INSTANCE := 'AV-35.05', RESTART :=, VISIBILITY :=, OPdwCmd :=, QdwState =>, QwState =>, QCLOSING =>, QCLOSE =>, QOPENING =>, QOPEN =>, QCMD_OP => "AV-35.05", QMON =>, QMON_ERR =>, QMON_T =>, QMON_T_CLOSE =>, QMAN_AUT =>, QREMOTE =>, QSIM =>, QLOCK =>, QERR =>, QERR_EXT =>, QwAlarm =>)
   END_RUNG
   RUNG wire#powerrail
      I_Contact( "AV-35.05" )
   END_RUNG wire#w1
   // the same network as SCL:
   #"AV-35.05"(LOCK := #lock,   // "Valve"
               LIOP_SEL := #Init,
               L_AUT := #Init,
               L_REMOTE := #Init,
               L_RESET := #Reset,
               FB_OPEN := "AV-35.05",
               FB_CLOSE := NOT "AV-35.05",
               L_MON := #Init,
               INSTANCE := 'AV-35.05',
               QCMD_OP => "AV-35.05");
END_REGION

REGION Network 66: AV-35.06
